REGION Network 1: Green
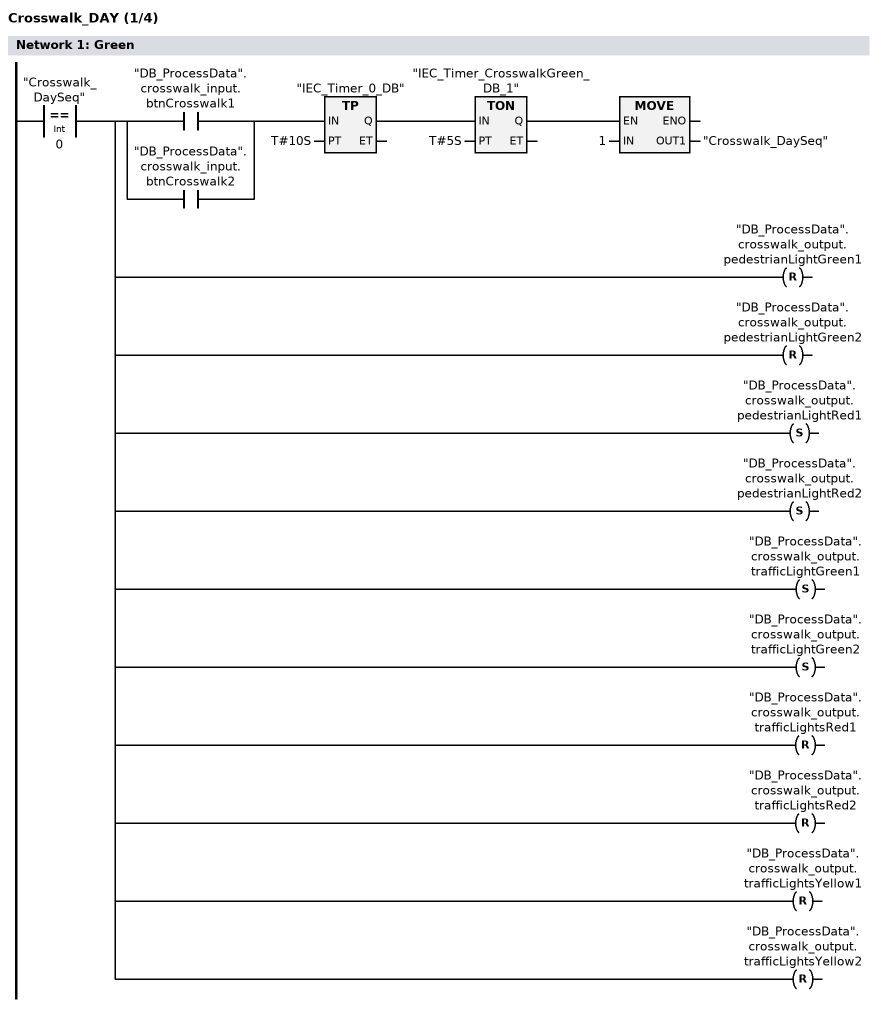
   #_w1 := "Crosswalk_DaySeq" = 0;
   "IEC_Timer_0_DB".TP(IN := #_w1 AND ("DB_ProcessData".crosswalk_input.btnCrosswalk1 OR "DB_ProcessData".crosswalk_input.btnCrosswalk2),
                       PT := T#10S);
   "IEC_Timer_CrosswalkGreen_DB_1".TON(IN := "IEC_Timer_0_DB".Q, PT := T#5S);
   IF "IEC_Timer_CrosswalkGreen_DB_1".Q THEN "Crosswalk_DaySeq" := 1; END_IF;
   IF #_w1 THEN
       "DB_ProcessData".crosswalk_output.pedestrianLightGreen1 := FALSE;
       "DB_ProcessData".crosswalk_output.pedestrianLightGreen2 := FALSE;
       "DB_ProcessData".crosswalk_output.pedestrianLightRed1 := TRUE;
       "DB_ProcessData".crosswalk_output.pedestrianLightRed2 := TRUE;
       "DB_ProcessData".crosswalk_output.trafficLightGreen1 := TRUE;
       "DB_ProcessData".crosswalk_output.trafficLightGreen2 := TRUE;
       "DB_ProcessData".crosswalk_output.trafficLightsRed1 := FALSE;
       "DB_ProcessData".crosswalk_output.trafficLightsRed2 := FALSE;
       "DB_ProcessData".crosswalk_output.trafficLightsYellow1 := FALSE;
       "DB_ProcessData".crosswalk_output.trafficLightsYellow2 := FALSE;
   END_IF;
END_REGION

REGION Network 2: Yellow1
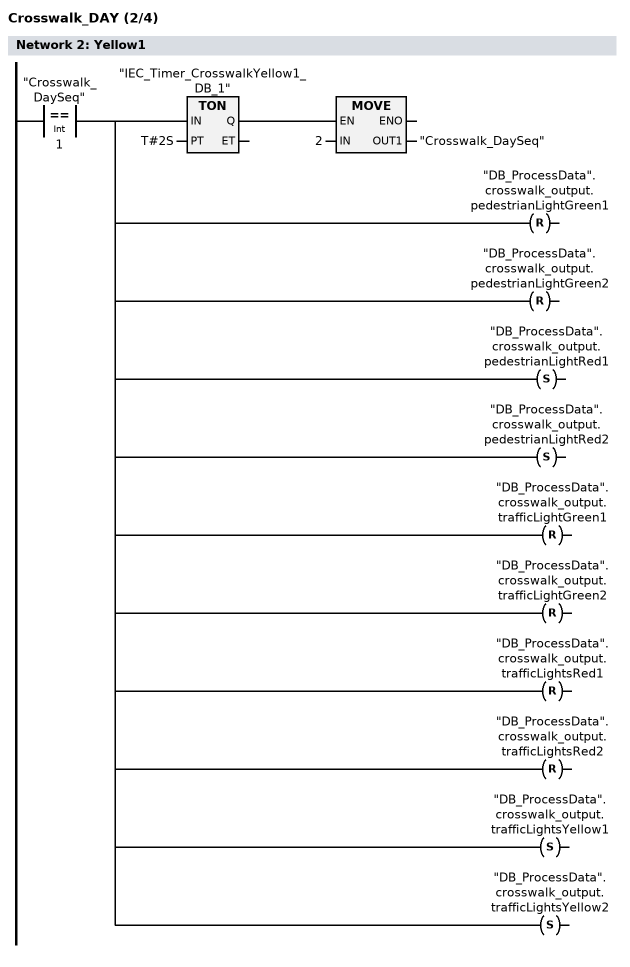
   #_w1 := "Crosswalk_DaySeq" = 1;
   "IEC_Timer_CrosswalkYellow1_DB_1".TON(IN := #_w1, PT := T#2S);
   IF "IEC_Timer_CrosswalkYellow1_DB_1".Q THEN "Crosswalk_DaySeq" := 2; END_IF;
   IF #_w1 THEN
       "DB_ProcessData".crosswalk_output.pedestrianLightGreen1 := FALSE;
       "DB_ProcessData".crosswalk_output.pedestrianLightGreen2 := FALSE;
       "DB_ProcessData".crosswalk_output.pedestrianLightRed1 := TRUE;
       "DB_ProcessData".crosswalk_output.pedestrianLightRed2 := TRUE;
       "DB_ProcessData".crosswalk_output.trafficLightGreen1 := FALSE;
       "DB_ProcessData".crosswalk_output.trafficLightGreen2 := FALSE;
       "DB_ProcessData".crosswalk_output.trafficLightsRed1 := FALSE;
       "DB_ProcessData".crosswalk_output.trafficLightsRed2 := FALSE;
       "DB_ProcessData".crosswalk_output.trafficLightsYellow1 := TRUE;
       "DB_ProcessData".crosswalk_output.trafficLightsYellow2 := TRUE;
   END_IF;
END_REGION

REGION Network 3: Red
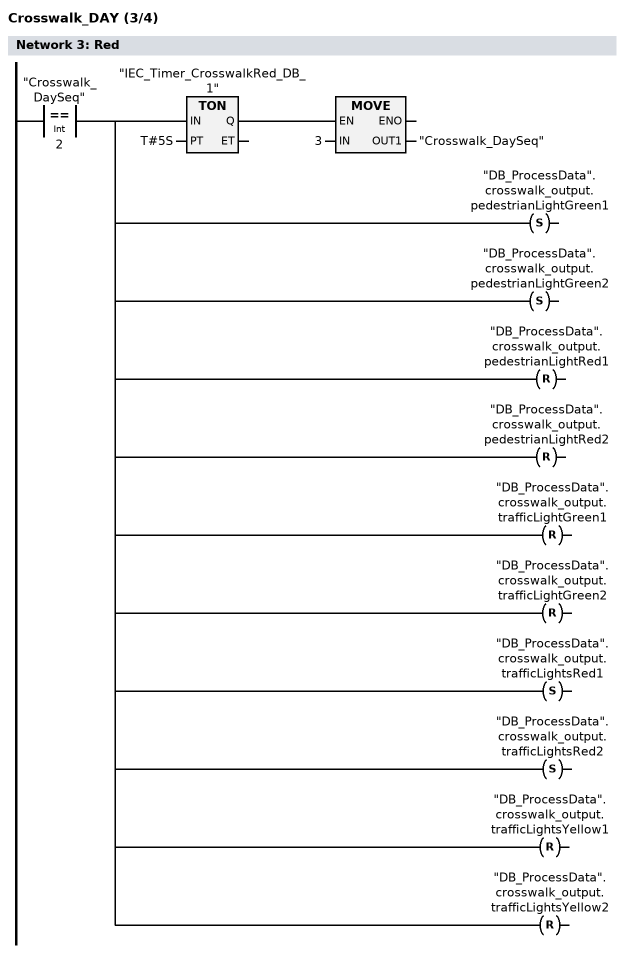
   #_w1 := "Crosswalk_DaySeq" = 2;
   "IEC_Timer_CrosswalkRed_DB_1".TON(IN := #_w1, PT := T#5S);
   IF "IEC_Timer_CrosswalkRed_DB_1".Q THEN "Crosswalk_DaySeq" := 3; END_IF;
   IF #_w1 THEN
       "DB_ProcessData".crosswalk_output.pedestrianLightGreen1 := TRUE;
       "DB_ProcessData".crosswalk_output.pedestrianLightGreen2 := TRUE;
       "DB_ProcessData".crosswalk_output.pedestrianLightRed1 := FALSE;
       "DB_ProcessData".crosswalk_output.pedestrianLightRed2 := FALSE;
       "DB_ProcessData".crosswalk_output.trafficLightGreen1 := FALSE;
       "DB_ProcessData".crosswalk_output.trafficLightGreen2 := FALSE;
       "DB_ProcessData".crosswalk_output.trafficLightsRed1 := TRUE;
       "DB_ProcessData".crosswalk_output.trafficLightsRed2 := TRUE;
       "DB_ProcessData".crosswalk_output.trafficLightsYellow1 := FALSE;
       "DB_ProcessData".crosswalk_output.trafficLightsYellow2 := FALSE;
   END_IF;
END_REGION

REGION Network 4: Yellow2
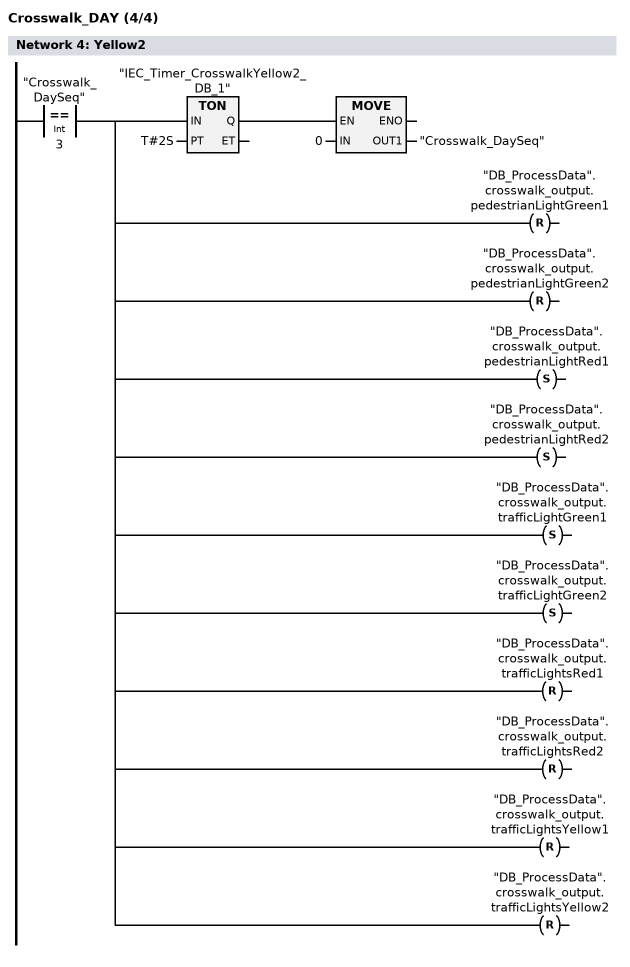
   #_w1 := "Crosswalk_DaySeq" = 3;
   "IEC_Timer_CrosswalkYellow2_DB_1".TON(IN := #_w1, PT := T#2S);
   IF "IEC_Timer_CrosswalkYellow2_DB_1".Q THEN "Crosswalk_DaySeq" := 0; END_IF;
   IF #_w1 THEN
       "DB_ProcessData".crosswalk_output.pedestrianLightGreen1 := FALSE;
       "DB_ProcessData".crosswalk_output.pedestrianLightGreen2 := FALSE;
       "DB_ProcessData".crosswalk_output.pedestrianLightRed1 := TRUE;
       "DB_ProcessData".crosswalk_output.pedestrianLightRed2 := TRUE;
       "DB_ProcessData".crosswalk_output.trafficLightGreen1 := TRUE;
       "DB_ProcessData".crosswalk_output.trafficLightGreen2 := TRUE;
       "DB_ProcessData".crosswalk_output.trafficLightsRed1 := FALSE;
       "DB_ProcessData".crosswalk_output.trafficLightsRed2 := FALSE;
       "DB_ProcessData".crosswalk_output.trafficLightsYellow1 := FALSE;
       "DB_ProcessData".crosswalk_output.trafficLightsYellow2 := FALSE;
   END_IF;
END_REGION
END_FUNCTION

FUNCTION "Crosswalk_NIGHT" : Void   // FC3, LAD
{ S7_Optimized_Access := 'TRUE' }
VERSION : 0.1
   VAR_TEMP   // added for the SCL form of the ladder/FBD networks
      _w1 : Bool;
   END_VAR
BEGIN

REGION Network 1: On
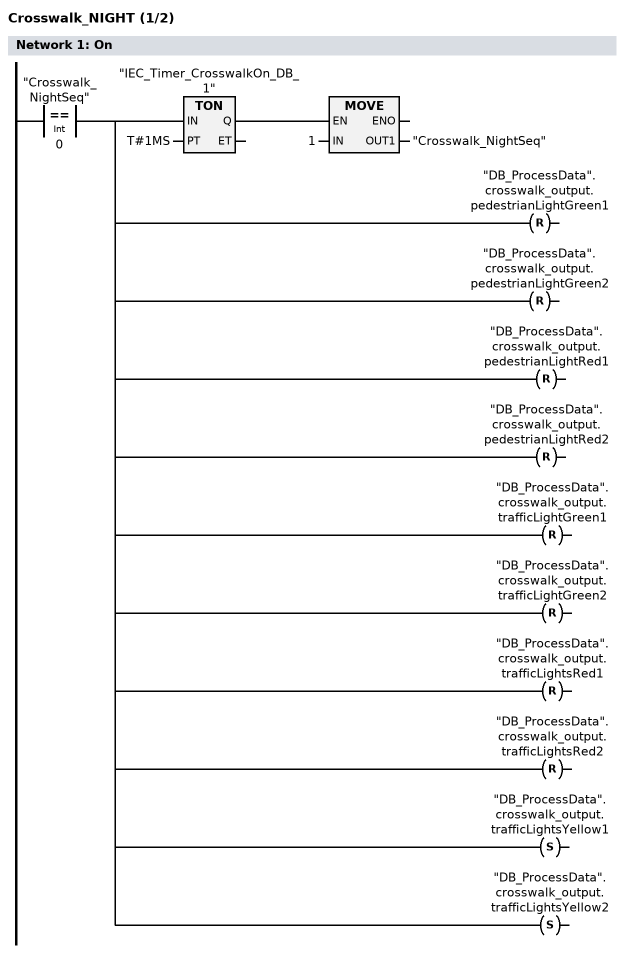
   #_w1 := "Crosswalk_NightSeq" = 0;
   "IEC_Timer_CrosswalkOn_DB_1".TON(IN := #_w1, PT := T#1MS);
   IF "IEC_Timer_CrosswalkOn_DB_1".Q THEN "Crosswalk_NightSeq" := 1; END_IF;
   IF #_w1 THEN
       "DB_ProcessData".crosswalk_output.pedestrianLightGreen1 := FALSE;
       "DB_ProcessData".crosswalk_output.pedestrianLightGreen2 := FALSE;
       "DB_ProcessData".crosswalk_output.pedestrianLightRed1 := FALSE;
       "DB_ProcessData".crosswalk_output.pedestrianLightRed2 := FALSE;
       "DB_ProcessData".crosswalk_output.trafficLightGreen1 := FALSE;
       "DB_ProcessData".crosswalk_output.trafficLightGreen2 := FALSE;
       "DB_ProcessData".crosswalk_output.trafficLightsRed1 := FALSE;
       "DB_ProcessData".crosswalk_output.trafficLightsRed2 := FALSE;
       "DB_ProcessData".crosswalk_output.trafficLightsYellow1 := TRUE;
       "DB_ProcessData".crosswalk_output.trafficLightsYellow2 := TRUE;
   END_IF;
END_REGION

REGION Network 2: Off
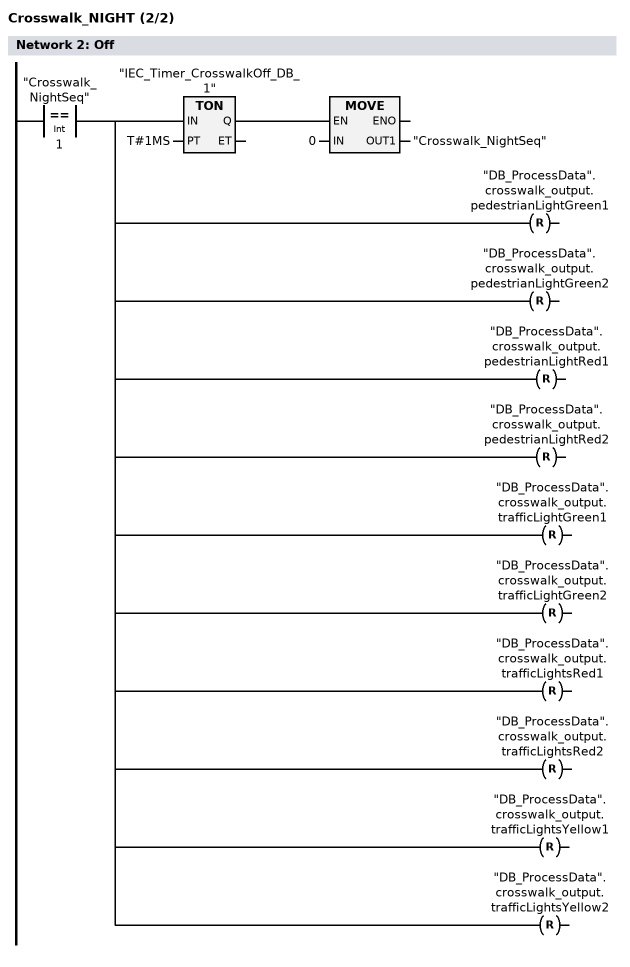
   #_w1 := "Crosswalk_NightSeq" = 1;
   "IEC_Timer_CrosswalkOff_DB_1".TON(IN := #_w1, PT := T#1MS);
   IF "IEC_Timer_CrosswalkOff_DB_1".Q THEN "Crosswalk_NightSeq" := 0; END_IF;
   IF #_w1 THEN
       "DB_ProcessData".crosswalk_output.pedestrianLightGreen1 := FALSE;
       "DB_ProcessData".crosswalk_output.pedestrianLightGreen2 := FALSE;
       "DB_ProcessData".crosswalk_output.pedestrianLightRed1 := FALSE;
       "DB_ProcessData".crosswalk_output.pedestrianLightRed2 := FALSE;
       "DB_ProcessData".crosswalk_output.trafficLightGreen1 := FALSE;
       "DB_ProcessData".crosswalk_output.trafficLightGreen2 := FALSE;
       "DB_ProcessData".crosswalk_output.trafficLightsRed1 := FALSE;
       "DB_ProcessData".crosswalk_output.trafficLightsRed2 := FALSE;
       "DB_ProcessData".crosswalk_output.trafficLightsYellow1 := FALSE;
       "DB_ProcessData".crosswalk_output.trafficLightsYellow2 := FALSE;
   END_IF;
END_REGION
END_FUNCTION

// folder: Regulator

FUNCTION "Regulator_PID" : Void   // FC5, LAD
{ S7_Optimized_Access := 'TRUE' }
VERSION : 0.1
BEGIN

REGION Network 1 (SCL)
   CASE "DB_ProcessData".regulator_input.order OF
       1:
           "Regulator_PV" := "DB_ProcessData".regulator_input.Uc1;
       2:
           "Regulator_PV" := "DB_ProcessData".regulator_input.Uc2;
       ELSE
           "Regulator_PV" := 0;
   END_CASE;

   "Regulator_SetPoint" := 50;
END_REGION

REGION Network 2
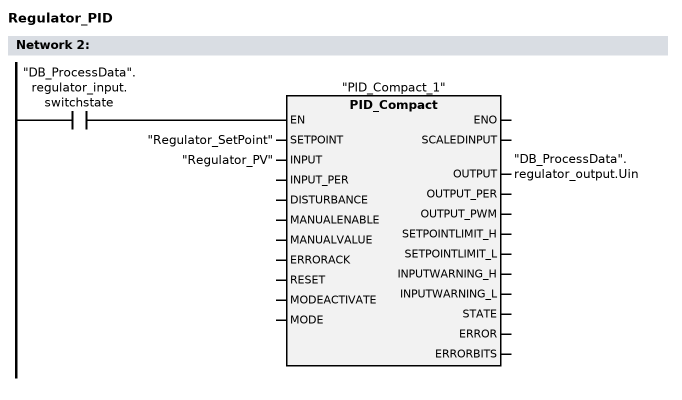
   IF "DB_ProcessData".regulator_input.switchstate THEN
       "PID_Compact_1"(Setpoint := "Regulator_SetPoint",   // PID_Compact
                       Input := "Regulator_PV",
                       Output => "DB_ProcessData".regulator_output.Uin);
   END_IF;
END_REGION
END_FUNCTION

// ===== PLC "R2D2_RESTAPI"  CPU 1212C DC/DC/DC =====

VAR_GLOBAL   // PLC tag table "Default tag table"
   "Clock_Byte" AT %MB0 : Byte;
   "Clock_10Hz" AT %M0.0 : Bool;
   "Clock_5Hz" AT %M0.1 : Bool;
   "Clock_2.5Hz" AT %M0.2 : Bool;
   "Clock_2Hz" AT %M0.3 : Bool;
   "Clock_1.25Hz" AT %M0.4 : Bool;
   "Clock_1Hz" AT %M0.5 : Bool;
   "Clock_0.625Hz" AT %M0.6 : Bool;
   "Clock_0.5Hz" AT %M0.7 : Bool;
   "System_Byte" AT %MB1 : Byte;
   "FirstScan" AT %M1.0 : Bool;
   "DiagStatusUpdate" AT %M1.1 : Bool;
   "AlwaysTRUE" AT %M1.2 : Bool;
   "AlwaysFALSE" AT %M1.3 : Bool;
END_VAR

VAR_GLOBAL   // PLC tag table "Regulator"
   "Regulator_PV" AT %MD100 : Real;
   "Regulator_SetPoint" AT %MD104 : Real;
END_VAR

VAR_GLOBAL   // PLC tag table "CarLight"
   "CarLight_Tag1" AT %I0.0 : Bool;
END_VAR

VAR_GLOBAL   // PLC tag table "Crossroad"
   "Crossroad_Tag_1" AT %M300.0 : Bool;
   "Crossroad_Tag_2" AT %M300.1 : Bool;
   "Crossroad_Tag_3" AT %MW302 : Word;
   "Crossroad_MEM 0" AT %M304.0 : Bool;
   "Crossroad_MEM 1" AT %M304.1 : Bool;
   "Crossroad_MEM 2" AT %M304.2 : Bool;
   "Crossroad_MEM 3" AT %M304.3 : Bool;
   "Crossroad_MEM 5" AT %M304.4 : Bool;
   "Crossroad_MEM 6" AT %M304.5 : Bool;
   "Crossroad_Clock" AT %MW328 : Int;
   "Crossroad_DayModeState" AT %MB305 : USInt;
   "Crossroad_ActualLengthState" AT %MD316 : Time;
   "Crossorad_HoursDayStart" AT %MW320 : Int;
   "Crossroad_HoursDayEnd" AT %MW322 : Int;
   "Crossroad_DayStarts" AT %MW324 : Int;
   "Crossroad_DayEnds" AT %MW326 : Int;
   "Crossroad_S1" AT %MB306 : USInt;
   "Crossroad_S2" AT %MB307 : USInt;
   "Crossroad_S3" AT %MB308 : USInt;
   "Crossroad_S4" AT %MB309 : USInt;
   "Crossroad_S5" AT %MB310 : USInt;
   "Crossroad_S6" AT %MB311 : USInt;
   "Crossroad_S7" AT %MB312 : USInt;
   "Crossroad_S8" AT %MB313 : USInt;
   "Crossroad_S9" AT %MB314 : USInt;
   "Crossroad_Walk_EN" AT %M330.0 : Bool;
END_VAR

VAR_GLOBAL   // PLC tag table "Crosswalk"
   "Crosswalk_CTU_current_value" AT %MW200 : Int;
   "Crosswalk_CTU_reset" AT %M202.0 : Bool;
   "Crosswalk_DayMode" AT %M202.1 : Bool;
   "Crosswalk_NightMode" AT %M202.2 : Bool;
   "Crosswalk_OffMode" AT %M202.3 : Bool;
   "Crosswalk_DaySeq" AT %MW204 : Int;
   "Crosswalk_NightSeq" AT %MW206 : Int;
END_VAR

TYPE "Crossroad_Input"
   STRUCT
      btnStart : Bool := FALSE;
      btnPause : Bool := FALSE;
      btnStop : Bool := FALSE;
      btnWestCrosswalk1 : Bool := FALSE;
      btnWestCrosswalk2 : Bool := FALSE;
      btnSouthCrosswalk1 : Bool := FALSE;
      btnSouthCrosswalk2 : Bool := FALSE;
      spare1 : DWord := 0;
      spare2 : DWord := 0;
      spare3 : DWord := 0;
      spare4 : DWord := 0;
   END_STRUCT;
END_TYPE

TYPE "Crossroad_Output"
   STRUCT
      crossroadType : Bool := FALSE;
      trafficLightNorth_green : Bool := FALSE;
      trafficLightNorth_yellow : Bool := FALSE;
      trafficLightNorth_red : Bool := FALSE;
      trafficLightSouth_green : Bool := FALSE;
      trafficLightSouth_yellow : Bool := FALSE;
      trafficLightSouth_red : Bool := FALSE;
      trafficLightWest_green : Bool := FALSE;
      trafficLightWest_yellow : Bool := FALSE;
      trafficLightWest_red : Bool := FALSE;
      trafficLightEast_green : Bool := FALSE;
      trafficLightEast_yellow : Bool := FALSE;
      trafficLightEast_red : Bool := FALSE;
      pedestrianSouth1_green : Bool := FALSE;
      pedestrianSouth1_red : Bool := FALSE;
      pedestrianSouth2_green : Bool := FALSE;
      pedestrianSouth2_red : Bool := FALSE;
      pedestrianWest1_green : Bool := FALSE;
      pedestrianWest1_red : Bool := FALSE;
      pedestrianWest2_green : Bool := FALSE;
      pedestrianWest2_red : Bool := FALSE;
      spare1 : DWord := 0;
      spare2 : DWord := 0;
      spare3 : DWord := 0;
      spare4 : DWord := 0;
   END_STRUCT;
END_TYPE

TYPE "Crosswalk_Input"
   STRUCT
      btnStart : Bool := FALSE;
      btnPause : Bool := FALSE;
      btnStop : Bool := FALSE;
      btnCrosswalk1 : Bool := FALSE;
      btnCrosswalk2 : Bool := FALSE;
      spare1 : DWord := 0;
      spare2 : DWord := 0;
      spare3 : DWord := 0;
      spare4 : DWord := 0;
   END_STRUCT;
END_TYPE

TYPE "Crosswalk_Output"
   STRUCT
      crosswalkType : Bool := FALSE;
      trafficLightGreen1 : Bool := FALSE;
      trafficLightsYellow1 : Bool := FALSE;
      trafficLightsRed1 : Bool := FALSE;
      trafficLightGreen2 : Bool := FALSE;
      trafficLightsYellow2 : Bool := FALSE;
      trafficLightsRed2 : Bool := FALSE;
      pedestrianLightGreen1 : Bool := FALSE;
      pedestrianLightRed1 : Bool := FALSE;
      pedestrianLightGreen2 : Bool := FALSE;
      pedestrianLightRed2 : Bool := FALSE;
      spare1 : DWord := 0;
      spare2 : DWord := 0;
      spare3 : DWord := 0;
      spare4 : DWord := 0;
   END_STRUCT;
END_TYPE

TYPE "Regulator_Input"
   STRUCT
      btnReset : Bool := FALSE;
      switchstate : Bool := FALSE;
      order : Int := 1;
      R1 : Real := 0.0;
      R2 : Real := 0.0;
      C1 : Real := 0.0;
      C2 : Real := 0.0;
      Uc1 : Real := 0.0;
      Uc2 : Real := 0.0;
      Td : Real := 0.0;
      Ts : Real := 0.0;
      spare1 : DWord := 0;
      spare2 : DWord := 0;
      spare3 : DWord := 0;
      spare4 : DWord := 0;
   END_STRUCT;
END_TYPE

TYPE "Regulator_Output"
   STRUCT
      Uin : Real := 0.0;
      spare1 : DWord := 0;
      spare2 : DWord := 0;
      spare3 : DWord := 0;
      spare4 : DWord := 0;
   END_STRUCT;
END_TYPE

TYPE "CarLight_Input"
   STRUCT
      btnReset : Bool := FALSE;
      error : Bool := FALSE;
      sensorLight : Bool := FALSE;
      sensorConnectorConnected : Bool := FALSE;
      result : Bool := FALSE;
      spare1 : DWord := 0;
      spare2 : DWord := 0;
      spare3 : DWord := 0;
      spare4 : DWord := 0;
   END_STRUCT;
END_TYPE

TYPE "CarLight_Output"
   STRUCT
      lowBeamLight : Bool := FALSE;
      highBeamLight : Bool := FALSE;
      turnLight : Bool := FALSE;
      spare1 : DWord := 0;
      spare2 : DWord := 0;
      spare3 : DWord := 0;
      spare4 : DWord := 0;
   END_STRUCT;
END_TYPE

// folder: Common

TYPE "typeDiagnostics"
TITLE = typeDiagnostics
// Provides a structure for detailed diagnostics
   STRUCT
      status : Word;   // Status of the block or error identification when error occurred
      subfunctionStatus : DWord;   // Status or return value of called FBs, FCs and system blocks
      stateNumber : DInt;   // State in the state machine of the block where the error occurred
   END_STRUCT;
END_TYPE

// folder: LHTTP

TYPE "LHTTP_typeTLS"
   STRUCT
      validateServerIdentity : Bool;   // Validate the subjectAlternateName in the X.509-V3 certificate of the server to check the identity of the server
      serverCert : UDInt;   // ID of the X.509-V3 certificate (usually a CA certificate) that is used by the TLS client to validate the TLS server authentication. If this parameter is 0, the TLS client uses all (CA) certificates currently loaded in the client certificate store to validate the server authentication.
      clientCert : UDInt;   // ID of own X.509 V3 certificate
   END_STRUCT;
END_TYPE

// folder: (top level)

DATA_BLOCK "DB_ProcessData"   // DB1
{ S7_Optimized_Access := 'TRUE' }
VERSION : 0.1
   VAR
      crossroad_input : "Crossroad_Input";
      crossroad_output : "Crossroad_Output";
      crosswalk_input : "Crosswalk_Input";
      crosswalk_output : "Crosswalk_Output";
      regulator_input : "Regulator_Input";
      regulator_output : "Regulator_Output";
      carlight_input : "CarLight_Input";
      carlight_output : "CarLight_Output";
   END_VAR
BEGIN
END_DATA_BLOCK

DATA_BLOCK "REST_API_DATA"   // DB2
{ S7_Optimized_Access := 'TRUE' }
VERSION : 0.1
   VAR
      DATA : Array[0..10000] of Char;
      REST_API_URL : String := 'http://192.168.1.101:5000/api/data';   // 'http://192.168.1.250:5000/api/data' + 'http://10.129.223.194:5000/api/data' + 'http://192.168.1.250:5000/api/data'
   END_VAR
BEGIN
END_DATA_BLOCK

DATA_BLOCK "LHTTP_PostPut_DB"   // DB13
{ S7_Optimized_Access := 'TRUE' }
AUTHOR : Siemens Industry Online Support
FAMILY : LHTTP
VERSION : 2.2
// stored: InstanceOfName LHTTP_PostPut
"LHTTP_PostPut"
BEGIN
END_DATA_BLOCK

DATA_BLOCK "LHTTP_Get_DB"   // DB14
{ S7_Optimized_Access := 'TRUE' }
AUTHOR : Siemens Industry Online Support
FAMILY : LHTTP
VERSION : 2.2
// stored: InstanceOfName LHTTP_Get
"LHTTP_Get"
BEGIN
END_DATA_BLOCK

// folder: CarLight

DATA_BLOCK "CarLight_SCL_DB"   // DB12
{ S7_Optimized_Access := 'TRUE' }
VERSION : 0.1
// stored: InstanceOfName CarLight_SCL
"CarLight_SCL"
BEGIN
END_DATA_BLOCK

// folder: System blocks/Program resources

DATA_BLOCK "IEC_Counter_0_DB"   // DB2
{ S7_Optimized_Access := 'TRUE' }
AUTHOR : Simatic
FAMILY : IEC
NAME : CNTR
VERSION : 1.0
// stored: InstanceOfName IEC_COUNTER
"IEC_COUNTER"
BEGIN
END_DATA_BLOCK

DATA_BLOCK "IEC_Timer_0_DB"   // DB3
{ S7_Optimized_Access := 'TRUE' }
AUTHOR : Simatic
FAMILY : IEC
NAME : IEC_TMR
VERSION : 1.0
// stored: InstanceOfName IEC_TIMER
"IEC_TIMER"
BEGIN
END_DATA_BLOCK

DATA_BLOCK "IEC_Timer_CrosswalkGreen_DB_1"   // DB4
{ S7_Optimized_Access := 'TRUE' }
AUTHOR : Simatic
FAMILY : IEC
NAME : IEC_TMR
VERSION : 1.0
// stored: InstanceOfName IEC_TIMER
"IEC_TIMER"
BEGIN
END_DATA_BLOCK

DATA_BLOCK "IEC_Timer_CrosswalkYellow1_DB_1"   // DB5
{ S7_Optimized_Access := 'TRUE' }
AUTHOR : Simatic
FAMILY : IEC
NAME : IEC_TMR
VERSION : 1.0
// stored: InstanceOfName IEC_TIMER
"IEC_TIMER"
BEGIN
END_DATA_BLOCK

DATA_BLOCK "IEC_Timer_CrosswalkRed_DB_1"   // DB6
{ S7_Optimized_Access := 'TRUE' }
AUTHOR : Simatic
FAMILY : IEC
NAME : IEC_TMR
VERSION : 1.0
// stored: InstanceOfName IEC_TIMER
"IEC_TIMER"
BEGIN
END_DATA_BLOCK

DATA_BLOCK "IEC_Timer_CrosswalkYellow2_DB_1"   // DB7
{ S7_Optimized_Access := 'TRUE' }
AUTHOR : Simatic
FAMILY : IEC
NAME : IEC_TMR
VERSION : 1.0
// stored: InstanceOfName IEC_TIMER
"IEC_TIMER"
BEGIN
END_DATA_BLOCK

DATA_BLOCK "IEC_Timer_CrosswalkOn_DB_1"   // DB8
{ S7_Optimized_Access := 'TRUE' }
AUTHOR : Simatic
FAMILY : IEC
NAME : IEC_TMR
VERSION : 1.0
// stored: InstanceOfName IEC_TIMER
"IEC_TIMER"
BEGIN
END_DATA_BLOCK

DATA_BLOCK "IEC_Timer_CrosswalkOff_DB_1"   // DB9
{ S7_Optimized_Access := 'TRUE' }
AUTHOR : Simatic
FAMILY : IEC
NAME : IEC_TMR
VERSION : 1.0
// stored: InstanceOfName IEC_TIMER
"IEC_TIMER"
BEGIN
END_DATA_BLOCK

DATA_BLOCK "IEC_Timer_CrossroadCycle_DB_1"   // DB10
{ S7_Optimized_Access := 'TRUE' }
AUTHOR : Simatic
FAMILY : IEC
NAME : IEC_TMR
VERSION : 1.0
// stored: InstanceOfName IEC_TIMER
"IEC_TIMER"
BEGIN
END_DATA_BLOCK

// folder: (top level)

ORGANIZATION_BLOCK "Main"   // OB1, LAD, ProgramCycle
TITLE = "Main Program Sweep (Cycle)"
{ S7_Optimized_Access := 'TRUE' }
VERSION : 0.1
   VAR_INPUT
      Initial_Call : Bool;   // Initial call of this OB
      Remanence : Bool;   // =True, if remanent data are available
   END_VAR
BEGIN

REGION Network 1: REST API - POST & GET
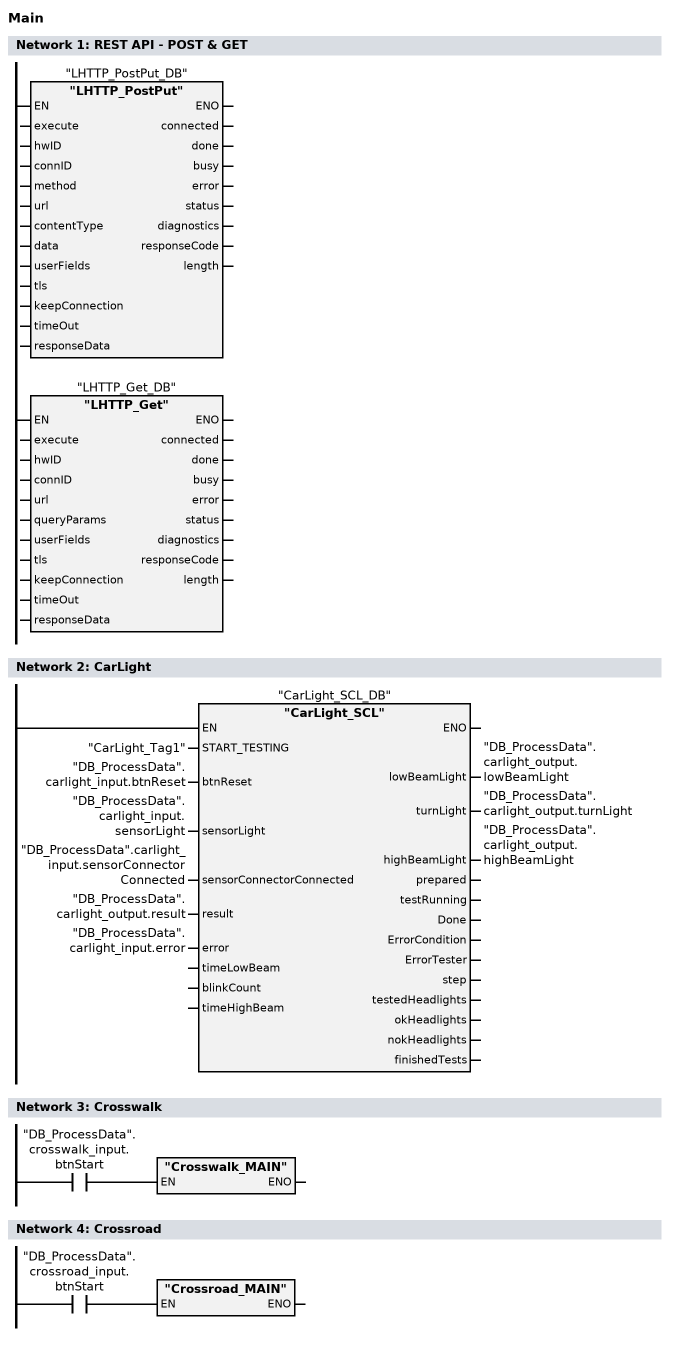
   RUNG wire#powerrail
      "LHTTP_PostPut_DB"(execute :=, hwID :=, connID :=, method :=, url :=, contentType :=, data :=, userFields :=, tls :=, keepConnection :=, timeOut :=, responseData :=, connected =>, done =>, busy =>, error =>, status =>, diagnostics =>, responseCode =>, length =>)
   END_RUNG
   RUNG wire#powerrail
      "LHTTP_Get_DB"(execute :=, hwID :=, connID :=, url :=, queryParams :=, userFields :=, tls :=, keepConnection :=, timeOut :=, responseData :=, connected =>, done =>, busy =>, error =>, status =>, diagnostics =>, responseCode =>, length =>)
   END_RUNG
   // the same network as SCL:
   "LHTTP_PostPut_DB"();   // "LHTTP_PostPut"
   "LHTTP_Get_DB"();   // "LHTTP_Get"
END_REGION

REGION Network 2: CarLight
   RUNG wire#powerrail
      "CarLight_SCL_DB"(START_TESTING := "CarLight_Tag1", btnReset := "DB_ProcessData".carlight_input.btnReset, sensorLight := "DB_ProcessData".carlight_input.sensorLight, sensorConnectorConnected := "DB_ProcessData".carlight_input.sensorConnectorConnected, result := "DB_ProcessData".carlight_output.result, error := "DB_ProcessData".carlight_input.error, timeLowBeam :=, blinkCount :=, timeHighBeam :=, lowBeamLight => "DB_ProcessData".carlight_output.lowBeamLight, turnLight => "DB_ProcessData".carlight_output.turnLight, highBeamLight => "DB_ProcessData".carlight_output.highBeamLight, prepared =>, testRunning =>, Done =>, ErrorCondition =>, ErrorTester =>, "step" =>, testedHeadlights =>, okHeadlights =>, nokHeadlights =>, finishedTests =>)
   END_RUNG
   // the same network as SCL:
   "CarLight_SCL_DB"(START_TESTING := "CarLight_Tag1",   // "CarLight_SCL"
                     btnReset := "DB_ProcessData".carlight_input.btnReset,
                     sensorLight := "DB_ProcessData".carlight_input.sensorLight,
                     sensorConnectorConnected := "DB_ProcessData".carlight_input.sensorConnectorConnected,
                     result := "DB_ProcessData".carlight_output.result,
                     error := "DB_ProcessData".carlight_input.error,
                     lowBeamLight => "DB_ProcessData".carlight_output.lowBeamLight,
                     turnLight => "DB_ProcessData".carlight_output.turnLight,
                     highBeamLight => "DB_ProcessData".carlight_output.highBeamLight);
END_REGION

REGION Network 3: Crosswalk
   RUNG wire#powerrail
      Contact( "DB_ProcessData".crosswalk_input.btnStart )
      "Crosswalk_MAIN"()
   END_RUNG
   // the same network as SCL:
   IF "DB_ProcessData".crosswalk_input.btnStart THEN "Crosswalk_MAIN"(); END_IF;
END_REGION

REGION Network 4: Crossroad
   RUNG wire#powerrail
      Contact( "DB_ProcessData".crossroad_input.btnStart )
      "Crossroad_MAIN"()
   END_RUNG
   // the same network as SCL:
   IF "DB_ProcessData".crossroad_input.btnStart THEN "Crossroad_MAIN"(); END_IF;
END_REGION
END_ORGANIZATION_BLOCK

ORGANIZATION_BLOCK "CyclicInterrupt"   // OB30, LAD, CyclicInterrupt
{ S7_Optimized_Access := 'TRUE' }
VERSION : 0.1
   VAR_INPUT
      Initial_Call : Bool;   // Initial call of this OB
      Event_Count : Int;   // Events discarded
   END_VAR
BEGIN

REGION Network 1: Regulator
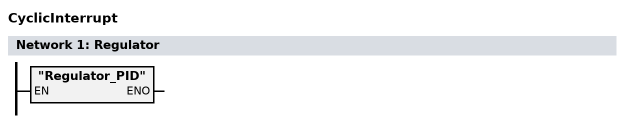
   RUNG wire#powerrail
      "Regulator_PID"()
   END_RUNG
   // the same network as SCL:
   "Regulator_PID"();
END_REGION
END_ORGANIZATION_BLOCK

ORGANIZATION_BLOCK "Startup"   // OB100, LAD, Startup
TITLE = "Complete Restart"
{ S7_Optimized_Access := 'TRUE' }
VERSION : 0.1
   VAR_INPUT
      LostRetentive : Bool;   // True if retentive data are lost
      LostRTC : Bool;   // True if date and time are lost
   END_VAR
BEGIN

REGION Network 1 (SCL)
   // Communication 


   // Crossroad
   "Crossorad_HoursDayStart" := 0;
   "Crossroad_HoursDayEnd" := 2400;
   "Crossroad_DayStarts" := 500;
   "Crossroad_DayEnds" := 2200;
   "Crossroad_S1" := 1;
   "Crossroad_S2" := 2;
   "Crossroad_S3" := 3;
   "Crossroad_S4" := 4;
   "Crossroad_S5" := 5;
   "Crossroad_S6" := 6;
   "Crossroad_S7" := 7;
   "Crossroad_S8" := 8;
   "Crossroad_S9" := 9;


   // Crosswalk


   // Regulaotr


   // CarLight
END_REGION
END_ORGANIZATION_BLOCK

// folder: CarLight

FUNCTION_BLOCK "CarLight_SCL"   // FB1, SCL
{ S7_Optimized_Access := 'TRUE' }
VERSION : 0.1
   VAR_INPUT
      START_TESTING : Bool;
      btnReset : Bool;
      sensorLight : Bool;
      sensorConnectorConnected : Bool;
      result : Bool;
      error : Bool;
      timeLowBeam : Time;
      blinkCount : Int;
      timeHighBeam : Time;
   END_VAR
   VAR_OUTPUT
      lowBeamLight : Bool;
      turnLight : Bool;
      highBeamLight : Bool;
      prepared : Bool;
      testRunning : Bool;
      Done : Bool;
      ErrorCondition : Bool;
      ErrorTester : Bool;
      "step" : Int;
      testedHeadlights : DInt;
      okHeadlights : DInt;
      nokHeadlights : DInt;
      finishedTests : DInt;
   END_VAR
   VAR
      state : Int;
      ready : Bool;
      start_old : Bool;
      start_rise : Bool;
      conditionsErrorLatched : Bool;
      testerErrorLatched : Bool;
      blinkTarget : Int;
      blinkIndex : Int;
      resultStored : Bool;
      testerResponseSeenTrue : Bool;
      tonLowBeam : TON_TIME;
      tonBlinkOn : TON_TIME;
      tonBlinkOff : TON_TIME;
      tonHighBeam : TON_TIME;
      tonAll : TON_TIME;
      tonTesterResponse : TON_TIME;
   END_VAR
BEGIN
   // ---------------------------------------------------------------------
   // Helper signals
   // ---------------------------------------------------------------------
   #ready := #sensorLight AND #sensorConnectorConnected;

   IF #blinkCount < 1 THEN
       #blinkTarget := 1;
   ELSE
       #blinkTarget := #blinkCount;
   END_IF;

   #start_rise := #START_TESTING AND NOT #start_old;
   #start_old := #START_TESTING;


   // ---------------------------------------------------------------------
   // RESET process (counters are NOT cleared)
   // ---------------------------------------------------------------------
   IF #btnReset THEN
       #state := 0;
       #conditionsErrorLatched := FALSE;
       #testerErrorLatched := FALSE;
       #blinkIndex := 0;
       #resultStored := FALSE;
       #testerResponseSeenTrue := FALSE;
   END_IF;


   // ---------------------------------------------------------------------
   // Loss of required conditions during test
   // ---------------------------------------------------------------------
   IF ((#state >= 20) AND (#state <= 55)) AND (NOT #ready) THEN
       #state := 0;
       #conditionsErrorLatched := TRUE;
       #blinkIndex := 0;
       #resultStored := FALSE;
       #testerResponseSeenTrue := FALSE;
   END_IF;


   // ---------------------------------------------------------------------
   // Tester error – immediate NOK termination
   // ---------------------------------------------------------------------
   IF ((#state >= 20) AND (#state <= 55)) AND #error THEN

       #testerErrorLatched := TRUE;

       IF NOT #resultStored THEN
           #testedHeadlights := #testedHeadlights + 1;
           #nokHeadlights := #nokHeadlights + 1;
           #resultStored := TRUE;
       END_IF;

       #blinkIndex := 0;
       #testerResponseSeenTrue := FALSE;

       #state := 70;

   END_IF;


   // ---------------------------------------------------------------------
   // State machine
   // ---------------------------------------------------------------------
   CASE #state OF


           // ==============================================================
           // 0 - IDLE
           // ==============================================================
       0:

           #lowBeamLight := FALSE;
           #turnLight := FALSE;
           #highBeamLight := FALSE;

           #tonLowBeam(IN := FALSE,
                     PT := #timeLowBeam);
           #tonBlinkOn(IN := FALSE,
                       PT := T#1s);
           #tonBlinkOff(IN := FALSE,
                        PT := T#1s);
           #tonHighBeam(IN := FALSE,
                     PT := #timeHighBeam);
           #tonAll(IN := FALSE,
                   PT := T#5s);
           #tonTesterResponse(IN := FALSE,
                              PT := T#1s);

           IF #start_rise THEN

               IF #ready AND (NOT #error) THEN

                   #conditionsErrorLatched := FALSE;
                   #testerErrorLatched := FALSE;
                   #blinkIndex := 0;
                   #resultStored := FALSE;
                   #testerResponseSeenTrue := FALSE;

                   #state := 20;

               ELSE

                   IF NOT #ready THEN
                       #conditionsErrorLatched := TRUE;
                   END_IF;

                   IF #error THEN
                       #testerErrorLatched := TRUE;
                   END_IF;

               END_IF;

           END_IF;


           // ==============================================================
           // 20 - LOW BEAM
           // ==============================================================
       20:

           #lowBeamLight := TRUE;
           #turnLight := FALSE;
           #highBeamLight := FALSE;

           #tonLowBeam(IN := TRUE,
                     PT := #timeLowBeam);
           #tonBlinkOn(IN := FALSE,
                       PT := T#1s);
           #tonBlinkOff(IN := FALSE,
                        PT := T#1s);
           #tonHighBeam(IN := FALSE,
                     PT := #timeHighBeam);
           #tonAll(IN := FALSE,
                   PT := T#5s);
           #tonTesterResponse(IN := FALSE,
                              PT := T#1s);

           IF #tonLowBeam.Q THEN
               #blinkIndex := 0;
               #state := 30;
           END_IF;


           // ==============================================================
           // 30 - TURN SIGNAL ON
           // ==============================================================
       30:

           #lowBeamLight := FALSE;
           #turnLight := TRUE;
           #highBeamLight := FALSE;

           #tonLowBeam(IN := FALSE,
                     PT := #timeLowBeam);
           #tonBlinkOn(IN := TRUE,
                       PT := T#1s);
           #tonBlinkOff(IN := FALSE,
                        PT := T#1s);
           #tonHighBeam(IN := FALSE,
                     PT := #timeHighBeam);
           #tonAll(IN := FALSE,
                   PT := T#5s);
           #tonTesterResponse(IN := FALSE,
                              PT := T#1s);

           IF #tonBlinkOn.Q THEN
               #state := 31;
           END_IF;


           // ==============================================================
           // 31 - TURN SIGNAL OFF
           // ==============================================================
       31:

           #lowBeamLight := FALSE;
           #turnLight := FALSE;
           #highBeamLight := FALSE;

           #tonLowBeam(IN := FALSE,
                     PT := #timeLowBeam);
           #tonBlinkOn(IN := FALSE,
                       PT := T#1s);
           #tonBlinkOff(IN := TRUE,
                        PT := T#1s);
           #tonHighBeam(IN := FALSE,
                     PT := #timeHighBeam);
           #tonAll(IN := FALSE,
                   PT := T#5s);
           #tonTesterResponse(IN := FALSE,
                              PT := T#1s);

           IF #tonBlinkOff.Q THEN

               #blinkIndex := #blinkIndex + 1;

               IF #blinkIndex < #blinkTarget THEN
                   #state := 30;
               ELSE
                   #state := 40;
               END_IF;

           END_IF;


           // ==============================================================
           // 40 - HIGH BEAM
           // ==============================================================
       40:

           #lowBeamLight := FALSE;
           #turnLight := FALSE;
           #highBeamLight := TRUE;

           #tonLowBeam(IN := FALSE,
                     PT := #timeLowBeam);
           #tonBlinkOn(IN := FALSE,
                       PT := T#1s);
           #tonBlinkOff(IN := FALSE,
                        PT := T#1s);
           #tonHighBeam(IN := TRUE,
                     PT := #timeHighBeam);
           #tonAll(IN := FALSE,
                   PT := T#5s);
           #tonTesterResponse(IN := FALSE,
                              PT := T#1s);

           IF #tonHighBeam.Q THEN
               #state := 50;
           END_IF;


           // ==============================================================
           // 50 - ALL LIGHTS (5 seconds)
           // ==============================================================
       50:

           #lowBeamLight := TRUE;
           #turnLight := TRUE;
           #highBeamLight := TRUE;

           #tonLowBeam(IN := FALSE,
                     PT := #timeLowBeam);
           #tonBlinkOn(IN := FALSE,
                       PT := T#1s);
           #tonBlinkOff(IN := FALSE,
                        PT := T#1s);
           #tonHighBeam(IN := FALSE,
                     PT := #timeHighBeam);
           #tonAll(IN := TRUE,
                   PT := T#5s);
           #tonTesterResponse(IN := FALSE,
                              PT := T#1s);

           IF #tonAll.Q THEN
               #testerResponseSeenTrue := FALSE;
               #state := 55;
           END_IF;


           // ==============================================================
           // 55 - WAIT 1 s FOR RESULT
           // ==============================================================
       55:

           #lowBeamLight := FALSE;
           #turnLight := FALSE;
           #highBeamLight := FALSE;

           #tonLowBeam(IN := FALSE,
                     PT := #timeLowBeam);
           #tonBlinkOn(IN := FALSE,
                       PT := T#1s);
           #tonBlinkOff(IN := FALSE,
                        PT := T#1s);
           #tonHighBeam(IN := FALSE,
                     PT := #timeHighBeam);
           #tonAll(IN := FALSE,
                   PT := T#5s);
           #tonTesterResponse(IN := TRUE,
                              PT := T#1s);

           IF #result THEN
               #testerResponseSeenTrue := TRUE;
           END_IF;

           IF #tonTesterResponse.Q THEN

               IF NOT #resultStored THEN

                   #testedHeadlights := #testedHeadlights + 1;

                   IF #testerResponseSeenTrue THEN
                       #okHeadlights := #okHeadlights + 1;
                   ELSE
                       #nokHeadlights := #nokHeadlights + 1;
                   END_IF;

                   #resultStored := TRUE;

               END_IF;

               #finishedTests := #finishedTests + 1;

               #state := 60;

           END_IF;


           // ==============================================================
           // 60 - FINISHED
           // ==============================================================
       60:

           #lowBeamLight := FALSE;
           #turnLight := FALSE;
           #highBeamLight := FALSE;

           IF #start_rise THEN

               IF #ready AND (NOT #error) THEN

                   #conditionsErrorLatched := FALSE;
                   #testerErrorLatched := FALSE;
                   #blinkIndex := 0;
                   #resultStored := FALSE;
                   #testerResponseSeenTrue := FALSE;

                   #state := 20;

               END_IF;

           END_IF;


           // ==============================================================
           // 70 - TESTER ERROR
           // ==============================================================
       70:

           #lowBeamLight := FALSE;
           #turnLight := FALSE;
           #highBeamLight := FALSE;

           IF #start_rise THEN

               IF #ready AND (NOT #error) THEN

                   #conditionsErrorLatched := FALSE;
                   #testerErrorLatched := FALSE;
                   #blinkIndex := 0;
                   #resultStored := FALSE;
                   #testerResponseSeenTrue := FALSE;

                   #state := 20;

               END_IF;

           END_IF;

       ELSE

           #state := 0;

   END_CASE;


   // ---------------------------------------------------------------------
   // State outputs
   // ---------------------------------------------------------------------
   #testRunning := (#state >= 20) AND (#state <= 55);

   #prepared := #ready AND (NOT #error) AND
   ((#state = 0) OR (#state = 60) OR (#state = 70));

   #Done := (#state = 60);

   #ErrorCondition := #conditionsErrorLatched;
   #ErrorTester := #testerErrorLatched;

   #step := #state;
END_FUNCTION_BLOCK

// folder: Common

FUNCTION "IsIPAddress" : Bool   // FC1, SCL
TITLE = IsIPAddress
{ S7_Optimized_Access := 'TRUE' }
VERSION : 0.1
// Evaluates whether a given String contains a valid IP address
   VAR_INPUT
      address : String;   // Address to be evaluated
   END_VAR
   VAR_OUTPUT
      ipAddress : IP_V4;   // Parsed IP address if passed address is IP address
   END_VAR
   VAR_TEMP
      tempAddress : String;   // Passed address
      tempOctet : String;   // Current octet
      tempIndex : DInt;   // Index for loop
      tempPos : Int;   // Position of found separator
      tempNum : Int;   // Converted octet
      tempIp : IP_V4;   // Parsed IP address
   END_VAR
   // Ret_Val : Return value
   VAR CONSTANT
      MAX_VALUE : USInt := 255;   // Max. valid value of octet
      NUM_OCTETS : DInt := 4;   // Number of octets
      CHAR_ZERO : Char := '0';   // ASCII character '0'
   END_VAR
BEGIN
   REGION BLOCK INFO HEADER
     //===============================================================================
     // SIEMENS / (c)Copyright 2024
     //-------------------------------------------------------------------------------
     // Title:        IsIPAddress
     // Function:     Evaluates whether a given String contains a valid IP address
     // Library:      --
     // Author:       Siemens Industry Online Support
     // Tested with:  CPU 1515-2 PN V3.1
     // Engineering:  TIA Portal V17
     // Restrictions: --
     // Requirements: S7-1200 with firmware V4.4 or higher
     //               S7-1500 with firmware V2.0 or higher
     //-------------------------------------------------------------------------------
     // Change log table:
     // Version  | Date       | Expert in charge       | Changes applied
     //-------------------------------------------------------------------------------
     // 01.00.00 | 2024-02-12 | Online Support         | First released version
     //===============================================================================
   END_REGION

   #tempAddress := #address;
   #IsIPAddress := FALSE; // Will be overwritten if IP address is detected
   #ipAddress := #tempIp; // Zero output parameter

   FOR #tempIndex := 1 TO #NUM_OCTETS DO
     #tempPos := FIND(IN1 := #tempAddress, IN2 := '.'); // Find separator

     IF (#tempPos > 0 OR #tempIndex = #NUM_OCTETS) // Separator found with exception of last octet
       AND NOT (#tempPos > 0 AND #tempIndex = #NUM_OCTETS) // No separator found in last octet
       AND #tempPos <= 4 // 3  characters or less
     THEN
       IF #tempIndex < #NUM_OCTETS THEN // First three octets
         #tempOctet := LEFT(IN := #tempAddress, L := #tempPos - 1);
       ELSE// Last octet
         #tempOctet := #tempAddress;
       END_IF;

       STRG_VAL(IN := #tempOctet,
                FORMAT := 0,
                P := 1,
                OUT => #tempNum);

       IF #tempNum >= 0 AND #tempNum <= #MAX_VALUE // Within 0 and 255
         AND NOT (#tempNum = 0 AND #tempIndex = 1) // Not 0 in first octet
         AND NOT (#tempNum = 0 AND #tempOctet[1] <> #CHAR_ZERO) // Not 0 because of invalid character
       THEN
         #tempIp.ADDR[#tempIndex] := INT_TO_BYTE(#tempNum);
         #tempAddress := RIGHT(IN := #tempAddress, L := LEN(#tempAddress) - #tempPos); // Remove evaluated octet
       ELSE // Address is not IP address
         EXIT;
       END_IF;
     ELSE // Address is not IP address
       EXIT;
     END_IF;

     IF #tempIndex = #NUM_OCTETS THEN // End of loop reached, address is IP address
       #ipAddress := #tempIp;
       #IsIPAddress := true;
     END_IF;
   END_FOR;
END_FUNCTION

// folder: Crossroad

FUNCTION "Crossroad_MAIN" : Void   // FC4, LAD
{ S7_Optimized_Access := 'TRUE' }
VERSION : 0.1
   VAR_TEMP   // added for the SCL form of the ladder/FBD networks
      _w1 : Bool;
      _w2 : Bool;
      _w3 : Bool;
      _w4 : Bool;
   END_VAR
BEGIN

REGION Network 1: Time based decision process
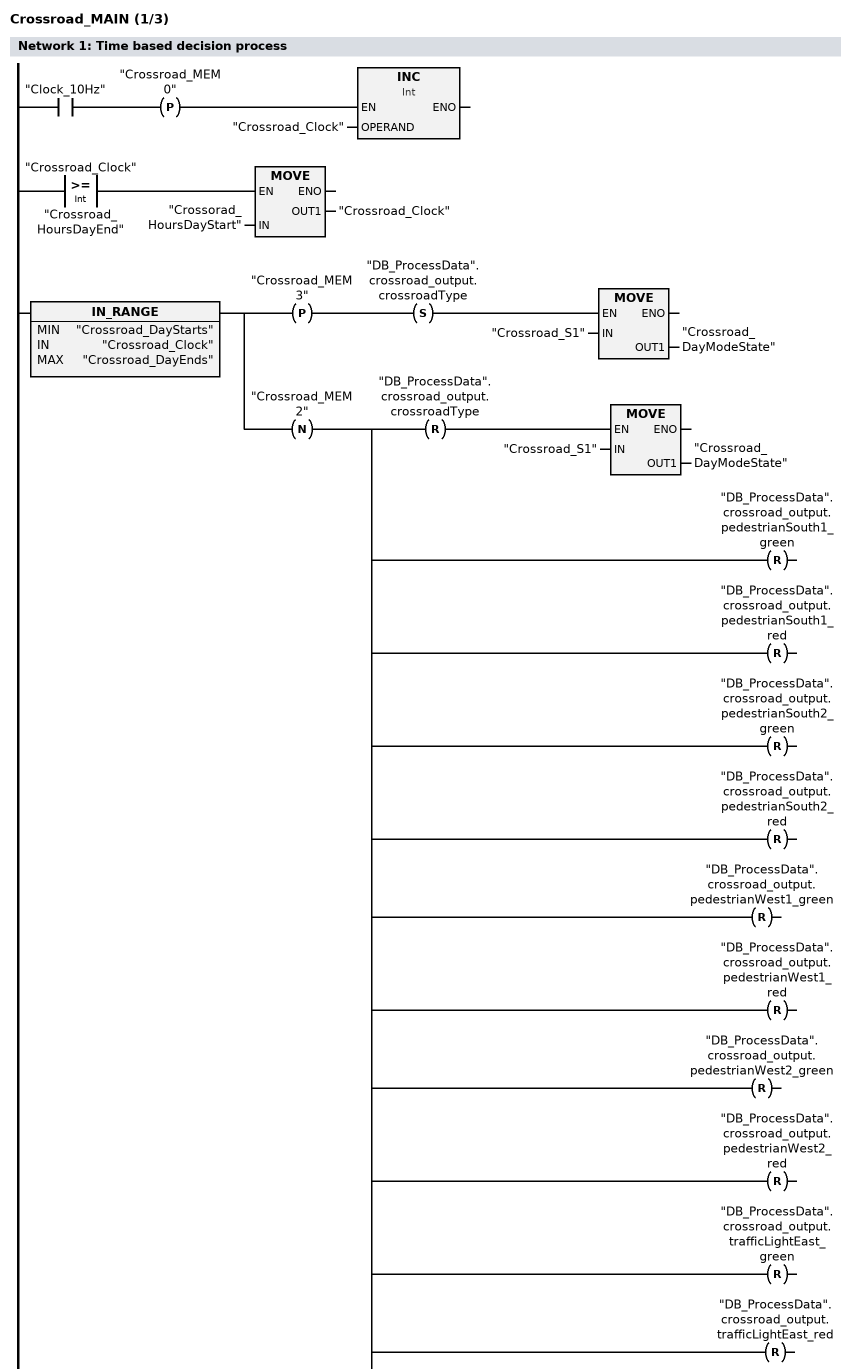
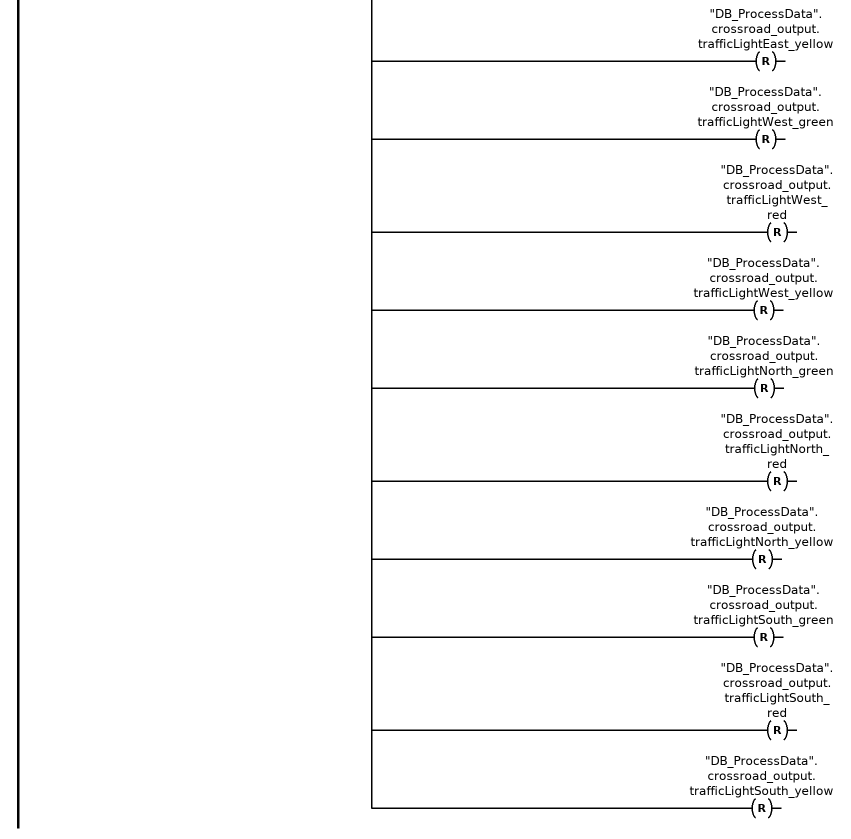
   RUNG wire#powerrail
      Contact( "Clock_10Hz" )
      P_Trig( "Crossroad_MEM 0" )
      { S7_Templates := "DestType := Int" } Inc( "Crossroad_Clock" )
   END_RUNG
   RUNG wire#powerrail
      { S7_Templates := "SrcType := Int" } GE_Contact(in1 := "Crossroad_Clock", in2 := "Crossroad_HoursDayEnd")
      Move(in := "Crossorad_HoursDayStart", out1 => "Crossroad_Clock")
   END_RUNG
   RUNG wire#powerrail
      { S7_Templates := "SrcType := Int" } InRange(min := "Crossroad_DayStarts", in := "Crossroad_Clock", max := "Crossroad_DayEnds")
      wire#w1
      P_Trig( "Crossroad_MEM 3" )
      S_Coil( "DB_ProcessData".crossroad_output.crossroadType )
      Move(in := "Crossroad_S1", out1 => "Crossroad_DayModeState")
   END_RUNG
   RUNG wire#w1
      N_Trig( "Crossroad_MEM 2" )
      wire#w2
      R_Coil( "DB_ProcessData".crossroad_output.crossroadType )
      Move(in := "Crossroad_S1", out1 => "Crossroad_DayModeState")
   END_RUNG
   RUNG wire#w2
      R_Coil( "DB_ProcessData".crossroad_output.pedestrianSouth1_green )
   END_RUNG
   RUNG wire#w2
      R_Coil( "DB_ProcessData".crossroad_output.pedestrianSouth1_red )
   END_RUNG
   RUNG wire#w2
      R_Coil( "DB_ProcessData".crossroad_output.pedestrianSouth2_green )
   END_RUNG
   RUNG wire#w2
      R_Coil( "DB_ProcessData".crossroad_output.pedestrianSouth2_red )
   END_RUNG
   RUNG wire#w2
      R_Coil( "DB_ProcessData".crossroad_output.pedestrianWest1_green )
   END_RUNG
   RUNG wire#w2
      R_Coil( "DB_ProcessData".crossroad_output.pedestrianWest1_red )
   END_RUNG
   RUNG wire#w2
      R_Coil( "DB_ProcessData".crossroad_output.pedestrianWest2_green )
   END_RUNG
   RUNG wire#w2
      R_Coil( "DB_ProcessData".crossroad_output.pedestrianWest2_red )
   END_RUNG
   RUNG wire#w2
      R_Coil( "DB_ProcessData".crossroad_output.trafficLightEast_green )
   END_RUNG
   RUNG wire#w2
      R_Coil( "DB_ProcessData".crossroad_output.trafficLightEast_red )
   END_RUNG
   RUNG wire#w2
      R_Coil( "DB_ProcessData".crossroad_output.trafficLightEast_yellow )
   END_RUNG
   RUNG wire#w2
      R_Coil( "DB_ProcessData".crossroad_output.trafficLightWest_green )
   END_RUNG
   RUNG wire#w2
      R_Coil( "DB_ProcessData".crossroad_output.trafficLightWest_red )
   END_RUNG
   RUNG wire#w2
      R_Coil( "DB_ProcessData".crossroad_output.trafficLightWest_yellow )
   END_RUNG
   RUNG wire#w2
      R_Coil( "DB_ProcessData".crossroad_output.trafficLightNorth_green )
   END_RUNG
   RUNG wire#w2
      R_Coil( "DB_ProcessData".crossroad_output.trafficLightNorth_red )
   END_RUNG
   RUNG wire#w2
      R_Coil( "DB_ProcessData".crossroad_output.trafficLightNorth_yellow )
   END_RUNG
   RUNG wire#w2
      R_Coil( "DB_ProcessData".crossroad_output.trafficLightSouth_green )
   END_RUNG
   RUNG wire#w2
      R_Coil( "DB_ProcessData".crossroad_output.trafficLightSouth_red )
   END_RUNG
   RUNG wire#w2
      R_Coil( "DB_ProcessData".crossroad_output.trafficLightSouth_yellow )
   END_RUNG
   // the same network as SCL:
   #_w1 := "Clock_10Hz" AND NOT "Crossroad_MEM 0";   // rising edge
   "Crossroad_MEM 0" := "Clock_10Hz";
   IF #_w1 THEN "Crossroad_Clock" := "Crossroad_Clock" + 1; END_IF;
   IF "Crossroad_Clock" >= "Crossroad_HoursDayEnd" THEN
       "Crossroad_Clock" := "Crossorad_HoursDayStart";
   END_IF;
   #_w2 := ("Crossroad_DayStarts" <= "Crossroad_Clock") AND ("Crossroad_Clock" <= "Crossroad_DayEnds");
   #_w3 := #_w2 AND NOT "Crossroad_MEM 3";   // rising edge
   "Crossroad_MEM 3" := #_w2;
   IF #_w3 THEN
       "DB_ProcessData".crossroad_output.crossroadType := TRUE;
       "Crossroad_DayModeState" := "Crossroad_S1";
   END_IF;
   #_w4 := NOT #_w2 AND "Crossroad_MEM 2";   // falling edge
   "Crossroad_MEM 2" := #_w2;
   IF #_w4 THEN
       "DB_ProcessData".crossroad_output.crossroadType := FALSE;
       "Crossroad_DayModeState" := "Crossroad_S1";
       "DB_ProcessData".crossroad_output.pedestrianSouth1_green := FALSE;
       "DB_ProcessData".crossroad_output.pedestrianSouth1_red := FALSE;
       "DB_ProcessData".crossroad_output.pedestrianSouth2_green := FALSE;
       "DB_ProcessData".crossroad_output.pedestrianSouth2_red := FALSE;
       "DB_ProcessData".crossroad_output.pedestrianWest1_green := FALSE;
       "DB_ProcessData".crossroad_output.pedestrianWest1_red := FALSE;
       "DB_ProcessData".crossroad_output.pedestrianWest2_green := FALSE;
       "DB_ProcessData".crossroad_output.pedestrianWest2_red := FALSE;
       "DB_ProcessData".crossroad_output.trafficLightEast_green := FALSE;
       "DB_ProcessData".crossroad_output.trafficLightEast_red := FALSE;
       "DB_ProcessData".crossroad_output.trafficLightEast_yellow := FALSE;
       "DB_ProcessData".crossroad_output.trafficLightWest_green := FALSE;
       "DB_ProcessData".crossroad_output.trafficLightWest_red := FALSE;
       "DB_ProcessData".crossroad_output.trafficLightWest_yellow := FALSE;
       "DB_ProcessData".crossroad_output.trafficLightNorth_green := FALSE;
       "DB_ProcessData".crossroad_output.trafficLightNorth_red := FALSE;
       "DB_ProcessData".crossroad_output.trafficLightNorth_yellow := FALSE;
       "DB_ProcessData".crossroad_output.trafficLightSouth_green := FALSE;
       "DB_ProcessData".crossroad_output.trafficLightSouth_red := FALSE;
       "DB_ProcessData".crossroad_output.trafficLightSouth_yellow := FALSE;
   END_IF;
END_REGION

REGION Network 2: Night mode
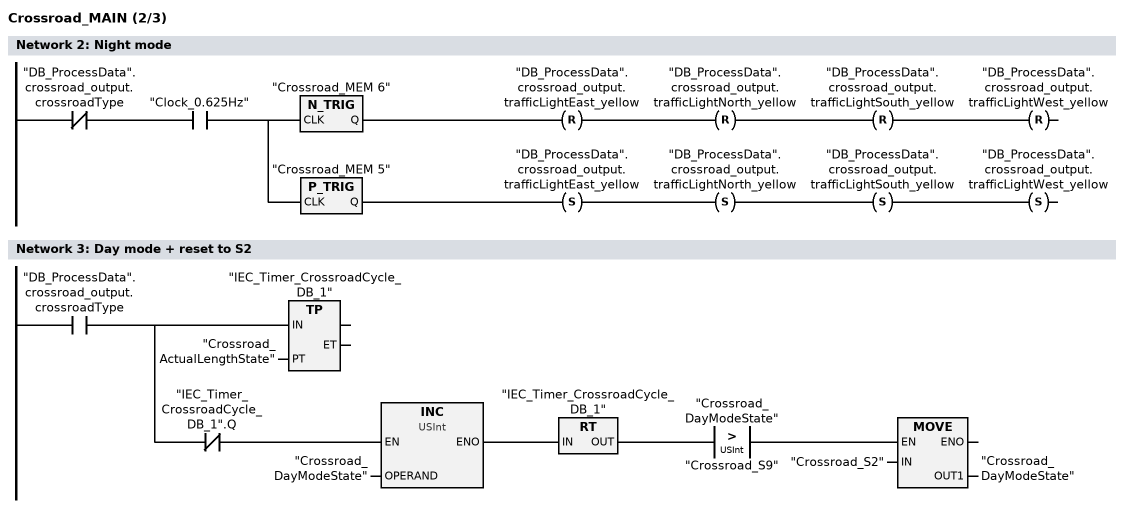
   RUNG wire#powerrail
      I_Contact( "DB_ProcessData".crossroad_output.crossroadType )
      Contact( "Clock_0.625Hz" )
      wire#w1
      N_Trig( "Crossroad_MEM 6" )
      R_Coil( "DB_ProcessData".crossroad_output.trafficLightEast_yellow )
      R_Coil( "DB_ProcessData".crossroad_output.trafficLightNorth_yellow )
      R_Coil( "DB_ProcessData".crossroad_output.trafficLightSouth_yellow )
      R_Coil( "DB_ProcessData".crossroad_output.trafficLightWest_yellow )
   END_RUNG
   RUNG wire#w1
      P_Trig( "Crossroad_MEM 5" )
      S_Coil( "DB_ProcessData".crossroad_output.trafficLightEast_yellow )
      S_Coil( "DB_ProcessData".crossroad_output.trafficLightNorth_yellow )
      S_Coil( "DB_ProcessData".crossroad_output.trafficLightSouth_yellow )
      S_Coil( "DB_ProcessData".crossroad_output.trafficLightWest_yellow )
   END_RUNG
   // the same network as SCL:
   #_w1 := NOT "DB_ProcessData".crossroad_output.crossroadType AND "Clock_0.625Hz";
   #_w2 := NOT #_w1 AND "Crossroad_MEM 6";   // falling edge
   "Crossroad_MEM 6" := #_w1;
   IF #_w2 THEN
       "DB_ProcessData".crossroad_output.trafficLightEast_yellow := FALSE;
       "DB_ProcessData".crossroad_output.trafficLightNorth_yellow := FALSE;
       "DB_ProcessData".crossroad_output.trafficLightSouth_yellow := FALSE;
       "DB_ProcessData".crossroad_output.trafficLightWest_yellow := FALSE;
   END_IF;
   #_w3 := #_w1 AND NOT "Crossroad_MEM 5";   // rising edge
   "Crossroad_MEM 5" := #_w1;
   IF #_w3 THEN
       "DB_ProcessData".crossroad_output.trafficLightEast_yellow := TRUE;
       "DB_ProcessData".crossroad_output.trafficLightNorth_yellow := TRUE;
       "DB_ProcessData".crossroad_output.trafficLightSouth_yellow := TRUE;
       "DB_ProcessData".crossroad_output.trafficLightWest_yellow := TRUE;
   END_IF;
END_REGION

REGION Network 3: Day mode + reset to S2
   "IEC_Timer_CrossroadCycle_DB_1".TP(IN := "DB_ProcessData".crossroad_output.crossroadType,
                           PT := "Crossroad_ActualLengthState");
   #_w1 := "DB_ProcessData".crossroad_output.crossroadType AND NOT "IEC_Timer_CrossroadCycle_DB_1".Q;
   IF #_w1 THEN
       "Crossroad_DayModeState" := "Crossroad_DayModeState" + 1;
       RESET_TIMER("IEC_Timer_CrossroadCycle_DB_1");
   END_IF;
   IF #_w1 AND ("Crossroad_DayModeState" > "Crossroad_S9") THEN
       "Crossroad_DayModeState" := "Crossroad_S2";
   END_IF;
END_REGION

REGION Network 4: Day mode time seq
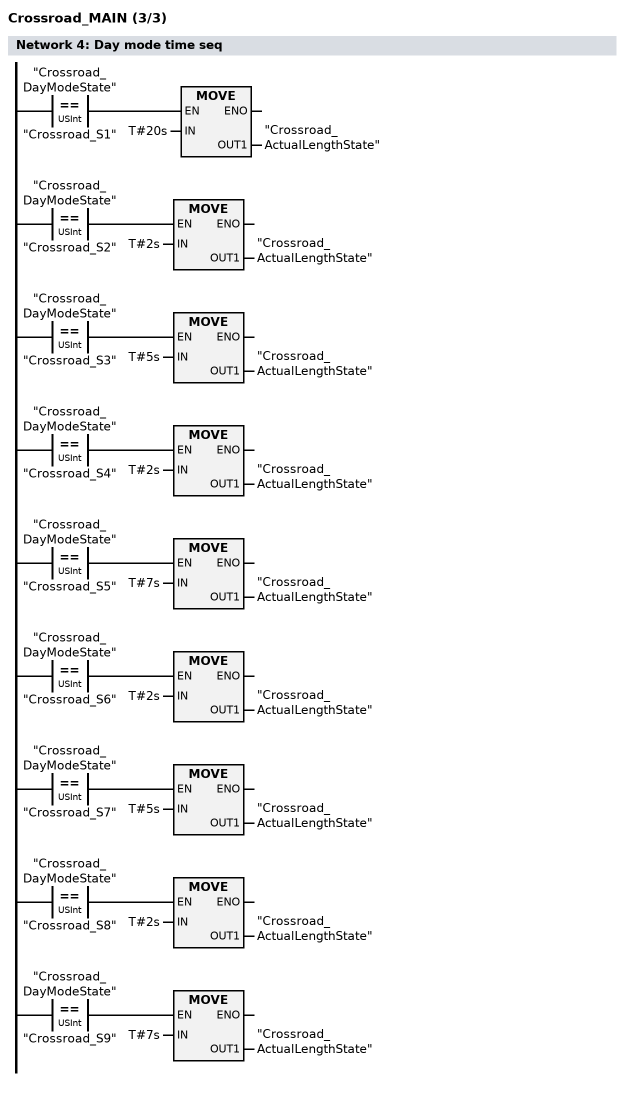
   RUNG wire#powerrail
      { S7_Templates := "SrcType := USInt" } EQ_Contact(in1 := "Crossroad_DayModeState", in2 := "Crossroad_S1")
      Move(in := T#20s, out1 => "Crossroad_ActualLengthState")
   END_RUNG
   RUNG wire#powerrail
      { S7_Templates := "SrcType := USInt" } EQ_Contact(in1 := "Crossroad_DayModeState", in2 := "Crossroad_S2")
      Move(in := T#2s, out1 => "Crossroad_ActualLengthState")
   END_RUNG
   RUNG wire#powerrail
      { S7_Templates := "SrcType := USInt" } EQ_Contact(in1 := "Crossroad_DayModeState", in2 := "Crossroad_S3")
      Move(in := T#5s, out1 => "Crossroad_ActualLengthState")
   END_RUNG
   RUNG wire#powerrail
      { S7_Templates := "SrcType := USInt" } EQ_Contact(in1 := "Crossroad_DayModeState", in2 := "Crossroad_S4")
      Move(in := T#2s, out1 => "Crossroad_ActualLengthState")
   END_RUNG
   RUNG wire#powerrail
      { S7_Templates := "SrcType := USInt" } EQ_Contact(in1 := "Crossroad_DayModeState", in2 := "Crossroad_S5")
      Move(in := T#7s, out1 => "Crossroad_ActualLengthState")
   END_RUNG
   RUNG wire#powerrail
      { S7_Templates := "SrcType := USInt" } EQ_Contact(in1 := "Crossroad_DayModeState", in2 := "Crossroad_S6")
      Move(in := T#2s, out1 => "Crossroad_ActualLengthState")
   END_RUNG
   RUNG wire#powerrail
      { S7_Templates := "SrcType := USInt" } EQ_Contact(in1 := "Crossroad_DayModeState", in2 := "Crossroad_S7")
      Move(in := T#5s, out1 => "Crossroad_ActualLengthState")
   END_RUNG
   RUNG wire#powerrail
      { S7_Templates := "SrcType := USInt" } EQ_Contact(in1 := "Crossroad_DayModeState", in2 := "Crossroad_S8")
      Move(in := T#2s, out1 => "Crossroad_ActualLengthState")
   END_RUNG
   RUNG wire#powerrail
      { S7_Templates := "SrcType := USInt" } EQ_Contact(in1 := "Crossroad_DayModeState", in2 := "Crossroad_S9")
      Move(in := T#7s, out1 => "Crossroad_ActualLengthState")
   END_RUNG
   // the same network as SCL:
   IF "Crossroad_DayModeState" = "Crossroad_S1" THEN "Crossroad_ActualLengthState" := T#20s; END_IF;
   IF "Crossroad_DayModeState" = "Crossroad_S2" THEN "Crossroad_ActualLengthState" := T#2s; END_IF;
   IF "Crossroad_DayModeState" = "Crossroad_S3" THEN "Crossroad_ActualLengthState" := T#5s; END_IF;
   IF "Crossroad_DayModeState" = "Crossroad_S4" THEN "Crossroad_ActualLengthState" := T#2s; END_IF;
   IF "Crossroad_DayModeState" = "Crossroad_S5" THEN "Crossroad_ActualLengthState" := T#7s; END_IF;
   IF "Crossroad_DayModeState" = "Crossroad_S6" THEN "Crossroad_ActualLengthState" := T#2s; END_IF;
   IF "Crossroad_DayModeState" = "Crossroad_S7" THEN "Crossroad_ActualLengthState" := T#5s; END_IF;
   IF "Crossroad_DayModeState" = "Crossroad_S8" THEN "Crossroad_ActualLengthState" := T#2s; END_IF;
   IF "Crossroad_DayModeState" = "Crossroad_S9" THEN "Crossroad_ActualLengthState" := T#7s; END_IF;
END_REGION

REGION Network 5 (SCL): Day mode lights
   IF "DB_ProcessData".crossroad_output.crossroadType THEN
       CASE "Crossroad_DayModeState" OF
           0:  // Statement section case S1
               // GREEN = FALSE, YELLOW = FALSE, RED = TRUE
               // PED: RED = TRUE, GREEN = FALSE

               "DB_ProcessData".crossroad_output.trafficLightEast_green := FALSE;
               "DB_ProcessData".crossroad_output.trafficLightEast_red := TRUE;
               "DB_ProcessData".crossroad_output.trafficLightEast_yellow := FALSE;

               "DB_ProcessData".crossroad_output.trafficLightNorth_green := FALSE;
               "DB_ProcessData".crossroad_output.trafficLightNorth_red := TRUE;
               "DB_ProcessData".crossroad_output.trafficLightNorth_yellow := FALSE;

               "DB_ProcessData".crossroad_output.trafficLightSouth_green := FALSE;
               "DB_ProcessData".crossroad_output.trafficLightSouth_red := TRUE;
               "DB_ProcessData".crossroad_output.trafficLightSouth_yellow := FALSE;

               "DB_ProcessData".crossroad_output.trafficLightWest_green := FALSE;
               "DB_ProcessData".crossroad_output.trafficLightWest_red := TRUE;
               "DB_ProcessData".crossroad_output.trafficLightWest_yellow := FALSE;

               "DB_ProcessData".crossroad_output.pedestrianSouth1_green := FALSE;
               "DB_ProcessData".crossroad_output.pedestrianSouth1_red := TRUE;
               "DB_ProcessData".crossroad_output.pedestrianSouth2_green := FALSE;
               "DB_ProcessData".crossroad_output.pedestrianSouth2_red := TRUE;

               "DB_ProcessData".crossroad_output.pedestrianWest1_green := FALSE;
               "DB_ProcessData".crossroad_output.pedestrianWest1_red := TRUE;
               "DB_ProcessData".crossroad_output.pedestrianWest2_green := FALSE;
               "DB_ProcessData".crossroad_output.pedestrianWest2_red := TRUE;

               //"PLC_LED_GREEN_1" := FALSE;
               //"PLC_LED_GREEN_2" := FALSE;
               //"PLC_LED_ORANGE_1" := FALSE;
               //"PLC_LED_ORANGE_2" := FALSE;
               //"PLC_LED_GREEN_CH" := FALSE;
               //"PLC_LED_RED_1" := TRUE;
               //"PLC_LED_RED_2" := TRUE;
               //"PLC_LED_RED_CH" := TRUE;

           1:  // Statement section case S2
               // GREEN = FALSE, RED = TRUE, YELLOW = TRUE
               // PED: RED = TRUE, GREEN = FALSE

               "DB_ProcessData".crossroad_output.trafficLightEast_green := FALSE;
               "DB_ProcessData".crossroad_output.trafficLightEast_red := TRUE;
               "DB_ProcessData".crossroad_output.trafficLightEast_yellow := TRUE;

               "DB_ProcessData".crossroad_output.trafficLightNorth_green := FALSE;
               "DB_ProcessData".crossroad_output.trafficLightNorth_red := TRUE;
               "DB_ProcessData".crossroad_output.trafficLightNorth_yellow := FALSE;

               "DB_ProcessData".crossroad_output.trafficLightSouth_green := FALSE;
               "DB_ProcessData".crossroad_output.trafficLightSouth_red := TRUE;
               "DB_ProcessData".crossroad_output.trafficLightSouth_yellow := FALSE;

               "DB_ProcessData".crossroad_output.trafficLightWest_green := FALSE;
               "DB_ProcessData".crossroad_output.trafficLightWest_red := TRUE;
               "DB_ProcessData".crossroad_output.trafficLightWest_yellow := TRUE;

               "DB_ProcessData".crossroad_output.pedestrianSouth1_green := FALSE;
               "DB_ProcessData".crossroad_output.pedestrianSouth1_red := TRUE;
               "DB_ProcessData".crossroad_output.pedestrianSouth2_green := FALSE;
               "DB_ProcessData".crossroad_output.pedestrianSouth2_red := TRUE;

               "DB_ProcessData".crossroad_output.pedestrianWest1_green := FALSE;
               "DB_ProcessData".crossroad_output.pedestrianWest1_red := TRUE;
               "DB_ProcessData".crossroad_output.pedestrianWest2_green := FALSE;
               "DB_ProcessData".crossroad_output.pedestrianWest2_red := TRUE;

               //"PLC_LED_GREEN_1" := FALSE;
               //"PLC_LED_GREEN_2" := FALSE;
               //"PLC_LED_ORANGE_1" := TRUE;
               //"PLC_LED_ORANGE_2" := FALSE;
               //"PLC_LED_GREEN_CH" := FALSE;
               //"PLC_LED_RED_1" := TRUE;
               //"PLC_LED_RED_2" := TRUE;
               //"PLC_LED_RED_CH" := TRUE;

           2:  // Statement section case S3
               // GREEN = TRUE, RED = FALSE, YELLOW = FALSE   // směr 1 (East, West)
               // GREEN = FALSE, RED = TRUE, YELLOW = FALSE   // směr 2 (North, South)
               // PED: RED = TRUE, GREEN = FALSE

               "DB_ProcessData".crossroad_output.trafficLightEast_green := TRUE;
               "DB_ProcessData".crossroad_output.trafficLightEast_red := FALSE;
               "DB_ProcessData".crossroad_output.trafficLightEast_yellow := FALSE;

               "DB_ProcessData".crossroad_output.trafficLightNorth_green := FALSE;
               "DB_ProcessData".crossroad_output.trafficLightNorth_red := TRUE;
               "DB_ProcessData".crossroad_output.trafficLightNorth_yellow := FALSE;

               "DB_ProcessData".crossroad_output.trafficLightSouth_green := FALSE;
               "DB_ProcessData".crossroad_output.trafficLightSouth_red := TRUE;
               "DB_ProcessData".crossroad_output.trafficLightSouth_yellow := FALSE;

               "DB_ProcessData".crossroad_output.trafficLightWest_green := TRUE;
               "DB_ProcessData".crossroad_output.trafficLightWest_red := FALSE;
               "DB_ProcessData".crossroad_output.trafficLightWest_yellow := FALSE;

               "DB_ProcessData".crossroad_output.pedestrianSouth1_green := FALSE;
               "DB_ProcessData".crossroad_output.pedestrianSouth1_red := TRUE;
               "DB_ProcessData".crossroad_output.pedestrianSouth2_green := FALSE;
               "DB_ProcessData".crossroad_output.pedestrianSouth2_red := TRUE;

               "DB_ProcessData".crossroad_output.pedestrianWest1_green := FALSE;
               "DB_ProcessData".crossroad_output.pedestrianWest1_red := TRUE;
               "DB_ProcessData".crossroad_output.pedestrianWest2_green := FALSE;
               "DB_ProcessData".crossroad_output.pedestrianWest2_red := TRUE;

               //"PLC_LED_GREEN_1" := TRUE;
               //"PLC_LED_GREEN_2" := FALSE;
               //"PLC_LED_ORANGE_1" := FALSE;
               //"PLC_LED_ORANGE_2" := FALSE;
               //"PLC_LED_GREEN_CH" := FALSE;
               //"PLC_LED_RED_1" := FALSE;
               //"PLC_LED_RED_2" := TRUE;
               //"PLC_LED_RED_CH" := TRUE;

           3:  // Statement section case S4
               // GREEN = FALSE, RED = FALSE, YELLOW = TRUE   // směr 1 (East, West)
               // GREEN = FALSE, RED = TRUE, YELLOW = FALSE   // směr 2 (North, South)
               // PED: RED = TRUE, GREEN = FALSE

               "DB_ProcessData".crossroad_output.trafficLightEast_green := FALSE;
               "DB_ProcessData".crossroad_output.trafficLightEast_red := FALSE;
               "DB_ProcessData".crossroad_output.trafficLightEast_yellow := TRUE;

               "DB_ProcessData".crossroad_output.trafficLightNorth_green := FALSE;
               "DB_ProcessData".crossroad_output.trafficLightNorth_red := TRUE;
               "DB_ProcessData".crossroad_output.trafficLightNorth_yellow := FALSE;

               "DB_ProcessData".crossroad_output.trafficLightSouth_green := FALSE;
               "DB_ProcessData".crossroad_output.trafficLightSouth_red := TRUE;
               "DB_ProcessData".crossroad_output.trafficLightSouth_yellow := FALSE;

               "DB_ProcessData".crossroad_output.trafficLightWest_green := FALSE;
               "DB_ProcessData".crossroad_output.trafficLightWest_red := FALSE;
               "DB_ProcessData".crossroad_output.trafficLightWest_yellow := TRUE;

               "DB_ProcessData".crossroad_output.pedestrianSouth1_green := FALSE;
               "DB_ProcessData".crossroad_output.pedestrianSouth1_red := TRUE;
               "DB_ProcessData".crossroad_output.pedestrianSouth2_green := FALSE;
               "DB_ProcessData".crossroad_output.pedestrianSouth2_red := TRUE;

               "DB_ProcessData".crossroad_output.pedestrianWest1_green := FALSE;
               "DB_ProcessData".crossroad_output.pedestrianWest1_red := TRUE;
               "DB_ProcessData".crossroad_output.pedestrianWest2_green := FALSE;
               "DB_ProcessData".crossroad_output.pedestrianWest2_red := TRUE;

               //"PLC_LED_GREEN_1" := FALSE;
               //"PLC_LED_GREEN_2" := FALSE;
               //"PLC_LED_ORANGE_1" := TRUE;
               //"PLC_LED_ORANGE_2" := FALSE;
               //"PLC_LED_GREEN_CH" := FALSE;
               //"PLC_LED_RED_1" := FALSE;
               //"PLC_LED_RED_2" := TRUE;
               //"PLC_LED_RED_CH" := TRUE;

           4:  // Statement section case S5
               // GREEN = FALSE, YELLOW = FALSE, RED = TRUE
               // PED: RED = TRUE, GREEN = FALSE

               "DB_ProcessData".crossroad_output.trafficLightEast_green := FALSE;
               "DB_ProcessData".crossroad_output.trafficLightEast_red := TRUE;
               "DB_ProcessData".crossroad_output.trafficLightEast_yellow := FALSE;

               "DB_ProcessData".crossroad_output.trafficLightNorth_green := FALSE;
               "DB_ProcessData".crossroad_output.trafficLightNorth_red := TRUE;
               "DB_ProcessData".crossroad_output.trafficLightNorth_yellow := FALSE;

               "DB_ProcessData".crossroad_output.trafficLightSouth_green := FALSE;
               "DB_ProcessData".crossroad_output.trafficLightSouth_red := TRUE;
               "DB_ProcessData".crossroad_output.trafficLightSouth_yellow := FALSE;

               "DB_ProcessData".crossroad_output.trafficLightWest_green := FALSE;
               "DB_ProcessData".crossroad_output.trafficLightWest_red := TRUE;
               "DB_ProcessData".crossroad_output.trafficLightWest_yellow := FALSE;

               "DB_ProcessData".crossroad_output.pedestrianSouth1_green := FALSE;
               "DB_ProcessData".crossroad_output.pedestrianSouth1_red := TRUE;
               "DB_ProcessData".crossroad_output.pedestrianSouth2_green := FALSE;
               "DB_ProcessData".crossroad_output.pedestrianSouth2_red := TRUE;

               "DB_ProcessData".crossroad_output.pedestrianWest1_green := FALSE;
               "DB_ProcessData".crossroad_output.pedestrianWest1_red := TRUE;
               "DB_ProcessData".crossroad_output.pedestrianWest2_green := FALSE;
               "DB_ProcessData".crossroad_output.pedestrianWest2_red := TRUE;

               //"PLC_LED_GREEN_1" := FALSE;
               //"PLC_LED_GREEN_2" := FALSE;
               //"PLC_LED_ORANGE_1" := FALSE;
               //"PLC_LED_ORANGE_2" := FALSE;
               //"PLC_LED_GREEN_CH" := FALSE;
               //"PLC_LED_RED_1" := TRUE;
               //"PLC_LED_RED_2" := TRUE;
               //"PLC_LED_RED_CH" := TRUE;

           5:  // Statement section case S6
               // GREEN = FALSE, RED = TRUE, YELLOW = FALSE   // směr 1 (East, West)
               // GREEN = FALSE, RED = TRUE, YELLOW = TRUE    // směr 2 (North, South)
               // PED: RED = TRUE, GREEN = FALSE (pokud není Crossroad_Walk_EN)

               "DB_ProcessData".crossroad_output.trafficLightEast_green := FALSE;
               "DB_ProcessData".crossroad_output.trafficLightEast_red := TRUE;
               "DB_ProcessData".crossroad_output.trafficLightEast_yellow := FALSE;

               "DB_ProcessData".crossroad_output.trafficLightNorth_green := FALSE;
               "DB_ProcessData".crossroad_output.trafficLightNorth_red := TRUE;
               "DB_ProcessData".crossroad_output.trafficLightNorth_yellow := TRUE;

               "DB_ProcessData".crossroad_output.trafficLightSouth_green := FALSE;
               "DB_ProcessData".crossroad_output.trafficLightSouth_red := TRUE;
               "DB_ProcessData".crossroad_output.trafficLightSouth_yellow := TRUE;

               "DB_ProcessData".crossroad_output.trafficLightWest_green := FALSE;
               "DB_ProcessData".crossroad_output.trafficLightWest_red := TRUE;
               "DB_ProcessData".crossroad_output.trafficLightWest_yellow := FALSE;

               "DB_ProcessData".crossroad_output.pedestrianSouth1_green := FALSE;
               "DB_ProcessData".crossroad_output.pedestrianSouth1_red := TRUE;
               "DB_ProcessData".crossroad_output.pedestrianSouth2_green := FALSE;
               "DB_ProcessData".crossroad_output.pedestrianSouth2_red := TRUE;

               "DB_ProcessData".crossroad_output.pedestrianWest1_green := FALSE;
               "DB_ProcessData".crossroad_output.pedestrianWest1_red := TRUE;
               "DB_ProcessData".crossroad_output.pedestrianWest2_green := FALSE;
               "DB_ProcessData".crossroad_output.pedestrianWest2_red := TRUE;

               //"PLC_LED_GREEN_1" := FALSE;
               //"PLC_LED_GREEN_2" := FALSE;
               //"PLC_LED_ORANGE_1" := FALSE;
               //"PLC_LED_ORANGE_2" := TRUE;
               //"PLC_LED_GREEN_CH" := FALSE;
               //"PLC_LED_RED_1" := TRUE;
               //"PLC_LED_RED_2" := TRUE;

               //"PLC_LED_GREEN_CH" := FALSE;
               //"PLC_LED_RED_CH" := TRUE;

               IF "Crossroad_Walk_EN" THEN
                   "DB_ProcessData".crossroad_output.pedestrianSouth1_green := TRUE;
                   "DB_ProcessData".crossroad_output.pedestrianSouth1_red := FALSE;
                   "DB_ProcessData".crossroad_output.pedestrianSouth2_green := TRUE;
                   "DB_ProcessData".crossroad_output.pedestrianSouth2_red := FALSE;

                   "DB_ProcessData".crossroad_output.pedestrianWest1_green := TRUE;
                   "DB_ProcessData".crossroad_output.pedestrianWest1_red := FALSE;
                   "DB_ProcessData".crossroad_output.pedestrianWest2_green := TRUE;
                   "DB_ProcessData".crossroad_output.pedestrianWest2_red := FALSE;

                   //"PLC_LED_GREEN_CH" := TRUE;
                   //"PLC_LED_RED_CH" := FALSE;
               END_IF;

           6:  // Statement section case S7
               // GREEN = FALSE, RED = TRUE, YELLOW = FALSE   // směr 1 (East, West)
               // GREEN = TRUE, RED = FALSE, YELLOW = FALSE   // směr 2 (North, South)
               // PED: RED = TRUE, GREEN = FALSE (pokud není Crossroad_Walk_EN)

               "DB_ProcessData".crossroad_output.trafficLightEast_green := FALSE;
               "DB_ProcessData".crossroad_output.trafficLightEast_red := TRUE;
               "DB_ProcessData".crossroad_output.trafficLightEast_yellow := FALSE;

               "DB_ProcessData".crossroad_output.trafficLightNorth_green := TRUE;
               "DB_ProcessData".crossroad_output.trafficLightNorth_red := FALSE;
               "DB_ProcessData".crossroad_output.trafficLightNorth_yellow := FALSE;

               "DB_ProcessData".crossroad_output.trafficLightSouth_green := TRUE;
               "DB_ProcessData".crossroad_output.trafficLightSouth_red := FALSE;
               "DB_ProcessData".crossroad_output.trafficLightSouth_yellow := FALSE;

               "DB_ProcessData".crossroad_output.trafficLightWest_green := FALSE;
               "DB_ProcessData".crossroad_output.trafficLightWest_red := TRUE;
               "DB_ProcessData".crossroad_output.trafficLightWest_yellow := FALSE;

               "DB_ProcessData".crossroad_output.pedestrianSouth1_green := FALSE;
               "DB_ProcessData".crossroad_output.pedestrianSouth1_red := TRUE;
               "DB_ProcessData".crossroad_output.pedestrianSouth2_green := FALSE;
               "DB_ProcessData".crossroad_output.pedestrianSouth2_red := TRUE;

               "DB_ProcessData".crossroad_output.pedestrianWest1_green := FALSE;
               "DB_ProcessData".crossroad_output.pedestrianWest1_red := TRUE;
               "DB_ProcessData".crossroad_output.pedestrianWest2_green := FALSE;
               "DB_ProcessData".crossroad_output.pedestrianWest2_red := TRUE;

               //"PLC_LED_GREEN_1" := FALSE;
               //"PLC_LED_GREEN_2" := TRUE;
               //"PLC_LED_ORANGE_1" := FALSE;
               //"PLC_LED_ORANGE_2" := FALSE;
               //"PLC_LED_RED_1" := TRUE;
               //"PLC_LED_RED_2" := FALSE;

               //"PLC_LED_GREEN_CH" := FALSE;
               //"PLC_LED_RED_CH" := TRUE;

               IF "Crossroad_Walk_EN" THEN
                   "DB_ProcessData".crossroad_output.pedestrianSouth1_green := TRUE;
                   "DB_ProcessData".crossroad_output.pedestrianSouth1_red := FALSE;
                   "DB_ProcessData".crossroad_output.pedestrianSouth2_green := TRUE;
                   "DB_ProcessData".crossroad_output.pedestrianSouth2_red := FALSE;

                   "DB_ProcessData".crossroad_output.pedestrianWest1_green := TRUE;
                   "DB_ProcessData".crossroad_output.pedestrianWest1_red := FALSE;
                   "DB_ProcessData".crossroad_output.pedestrianWest2_green := TRUE;
                   "DB_ProcessData".crossroad_output.pedestrianWest2_red := FALSE;

                   //"PLC_LED_GREEN_CH" := TRUE;
                   //"PLC_LED_RED_CH" := FALSE;
               END_IF;

           7:  // Statement section case S8
               // GREEN = FALSE, RED = TRUE, YELLOW = FALSE   // směr 1 (East, West)
               // GREEN = FALSE, RED = FALSE, YELLOW = TRUE   // směr 2 (North, South)
               // PED: RED = TRUE, GREEN = FALSE

               "DB_ProcessData".crossroad_output.trafficLightEast_green := FALSE;
               "DB_ProcessData".crossroad_output.trafficLightEast_red := TRUE;
               "DB_ProcessData".crossroad_output.trafficLightEast_yellow := FALSE;

               "DB_ProcessData".crossroad_output.trafficLightNorth_green := FALSE;
               "DB_ProcessData".crossroad_output.trafficLightNorth_red := FALSE;
               "DB_ProcessData".crossroad_output.trafficLightNorth_yellow := TRUE;

               "DB_ProcessData".crossroad_output.trafficLightSouth_green := FALSE;
               "DB_ProcessData".crossroad_output.trafficLightSouth_red := FALSE;
               "DB_ProcessData".crossroad_output.trafficLightSouth_yellow := TRUE;

               "DB_ProcessData".crossroad_output.trafficLightWest_green := FALSE;
               "DB_ProcessData".crossroad_output.trafficLightWest_red := TRUE;
               "DB_ProcessData".crossroad_output.trafficLightWest_yellow := FALSE;

               "DB_ProcessData".crossroad_output.pedestrianSouth1_green := FALSE;
               "DB_ProcessData".crossroad_output.pedestrianSouth1_red := TRUE;
               "DB_ProcessData".crossroad_output.pedestrianSouth2_green := FALSE;
               "DB_ProcessData".crossroad_output.pedestrianSouth2_red := TRUE;

               "DB_ProcessData".crossroad_output.pedestrianWest1_green := FALSE;
               "DB_ProcessData".crossroad_output.pedestrianWest1_red := TRUE;
               "DB_ProcessData".crossroad_output.pedestrianWest2_green := FALSE;
               "DB_ProcessData".crossroad_output.pedestrianWest2_red := TRUE;

               //"PLC_LED_GREEN_1" := FALSE;
               //"PLC_LED_GREEN_2" := FALSE;
               //"PLC_LED_ORANGE_1" := FALSE;
               //"PLC_LED_ORANGE_2" := TRUE;
               //"PLC_LED_GREEN_CH" := FALSE;
               //"PLC_LED_RED_1" := TRUE;
               //"PLC_LED_RED_2" := FALSE;
               //"PLC_LED_RED_CH" := TRUE;

           8:  // Statement section case S9
               // GREEN = FALSE, YELLOW = FALSE, RED = TRUE
               // PED: RED = TRUE, GREEN = FALSE

               "DB_ProcessData".crossroad_output.trafficLightEast_green := FALSE;
               "DB_ProcessData".crossroad_output.trafficLightEast_red := TRUE;
               "DB_ProcessData".crossroad_output.trafficLightEast_yellow := FALSE;

               "DB_ProcessData".crossroad_output.trafficLightNorth_green := FALSE;
               "DB_ProcessData".crossroad_output.trafficLightNorth_red := TRUE;
               "DB_ProcessData".crossroad_output.trafficLightNorth_yellow := FALSE;

               "DB_ProcessData".crossroad_output.trafficLightSouth_green := FALSE;
               "DB_ProcessData".crossroad_output.trafficLightSouth_red := TRUE;
               "DB_ProcessData".crossroad_output.trafficLightSouth_yellow := FALSE;

               "DB_ProcessData".crossroad_output.trafficLightWest_green := FALSE;
               "DB_ProcessData".crossroad_output.trafficLightWest_red := TRUE;
               "DB_ProcessData".crossroad_output.trafficLightWest_yellow := FALSE;

               "DB_ProcessData".crossroad_output.pedestrianSouth1_green := FALSE;
               "DB_ProcessData".crossroad_output.pedestrianSouth1_red := TRUE;
               "DB_ProcessData".crossroad_output.pedestrianSouth2_green := FALSE;
               "DB_ProcessData".crossroad_output.pedestrianSouth2_red := TRUE;

               "DB_ProcessData".crossroad_output.pedestrianWest1_green := FALSE;
               "DB_ProcessData".crossroad_output.pedestrianWest1_red := TRUE;
               "DB_ProcessData".crossroad_output.pedestrianWest2_green := FALSE;
               "DB_ProcessData".crossroad_output.pedestrianWest2_red := TRUE;

               //"PLC_LED_GREEN_1" := FALSE;
               //"PLC_LED_GREEN_2" := FALSE;
               //"PLC_LED_ORANGE_1" := FALSE;
               //"PLC_LED_ORANGE_2" := FALSE;
               //"PLC_LED_GREEN_CH" := FALSE;
               //"PLC_LED_RED_1" := TRUE;
               //"PLC_LED_RED_2" := TRUE;
               //"PLC_LED_RED_CH" := TRUE;

               "Crossroad_Walk_EN" := FALSE;

           ELSE  // Statement section ELSE
               "DB_ProcessData".crossroad_output.trafficLightEast_green := FALSE;
               "DB_ProcessData".crossroad_output.trafficLightEast_red := FALSE;
               "DB_ProcessData".crossroad_output.trafficLightEast_yellow := FALSE;

               "DB_ProcessData".crossroad_output.trafficLightNorth_green := FALSE;
               "DB_ProcessData".crossroad_output.trafficLightNorth_red := FALSE;
               "DB_ProcessData".crossroad_output.trafficLightNorth_yellow := FALSE;

               "DB_ProcessData".crossroad_output.trafficLightSouth_green := FALSE;
               "DB_ProcessData".crossroad_output.trafficLightSouth_red := FALSE;
               "DB_ProcessData".crossroad_output.trafficLightSouth_yellow := FALSE;

               "DB_ProcessData".crossroad_output.trafficLightWest_green := FALSE;
               "DB_ProcessData".crossroad_output.trafficLightWest_red := FALSE;
               "DB_ProcessData".crossroad_output.trafficLightWest_yellow := FALSE;

               "DB_ProcessData".crossroad_output.pedestrianSouth1_green := FALSE;
               "DB_ProcessData".crossroad_output.pedestrianSouth1_red := FALSE;
               "DB_ProcessData".crossroad_output.pedestrianSouth2_green := FALSE;
               "DB_ProcessData".crossroad_output.pedestrianSouth2_red := FALSE;

               "DB_ProcessData".crossroad_output.pedestrianWest1_green := FALSE;
               "DB_ProcessData".crossroad_output.pedestrianWest1_red := FALSE;
               "DB_ProcessData".crossroad_output.pedestrianWest2_green := FALSE;
               "DB_ProcessData".crossroad_output.pedestrianWest2_red := FALSE;

               //"PLC_LED_GREEN_1" := FALSE;
               //"PLC_LED_GREEN_2" := FALSE;
               //"PLC_LED_ORANGE_1" := FALSE;
               //"PLC_LED_ORANGE_2" := FALSE;
               //"PLC_LED_RED_1" := FALSE;
               //"PLC_LED_RED_2" := FALSE;
               //"PLC_LED_GREEN_CH" := FALSE;
               //"PLC_LED_RED_CH" := FALSE;

               "Crossroad_Walk_EN" := FALSE;
       END_CASE;
   END_IF;
END_REGION

REGION Network 6 (SCL): Pedestrians bnts
   IF "DB_ProcessData".crossroad_input.btnSouthCrosswalk1 OR "DB_ProcessData".crossroad_input.btnSouthCrosswalk2 OR "DB_ProcessData".crossroad_input.btnWestCrosswalk1 OR "DB_ProcessData".crossroad_input.btnWestCrosswalk2 THEN
       "Crossroad_Walk_EN" := TRUE;
   END_IF;
END_REGION
END_FUNCTION

// folder: Crosswalk

FUNCTION "Crosswalk_MAIN" : Void   // FC1, LAD
{ S7_Optimized_Access := 'TRUE' }
VERSION : 0.1
BEGIN

REGION Network 1: Control
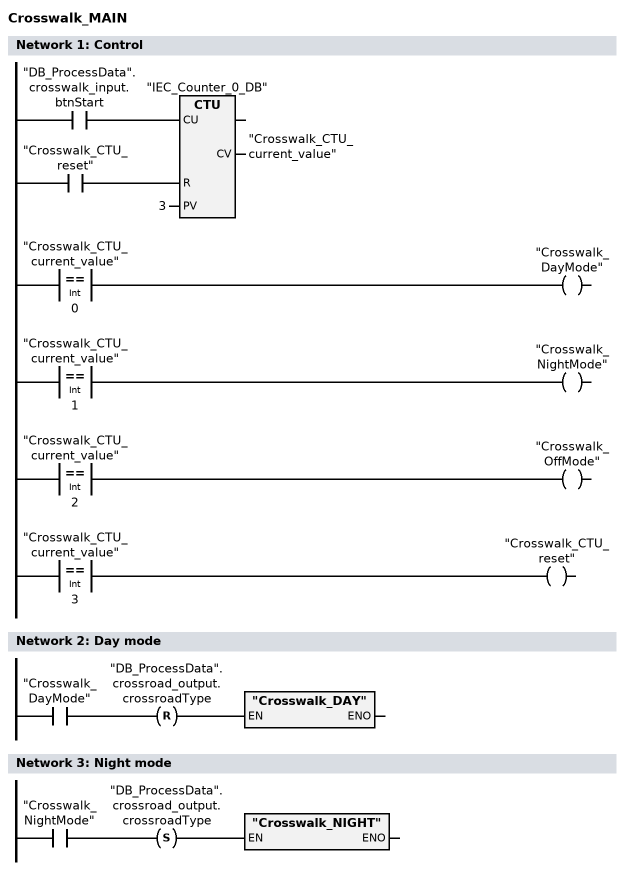
   "IEC_Counter_0_DB".CTU(CU := "DB_ProcessData".crosswalk_input.btnStart,
                          R := "Crosswalk_CTU_reset",
                          PV := 3,
                          CV => "Crosswalk_CTU_current_value");
   "Crosswalk_DayMode" := "Crosswalk_CTU_current_value" = 0;
   "Crosswalk_NightMode" := "Crosswalk_CTU_current_value" = 1;
   "Crosswalk_OffMode" := "Crosswalk_CTU_current_value" = 2;
   "Crosswalk_CTU_reset" := "Crosswalk_CTU_current_value" = 3;
END_REGION

REGION Network 2: Day mode
   RUNG wire#powerrail
      Contact( "Crosswalk_DayMode" )
      R_Coil( "DB_ProcessData".crossroad_output.crossroadType )
      "Crosswalk_DAY"()
   END_RUNG
   // the same network as SCL:
   IF "Crosswalk_DayMode" THEN
       "DB_ProcessData".crossroad_output.crossroadType := FALSE;
       "Crosswalk_DAY"();
   END_IF;
END_REGION

REGION Network 3: Night mode
   RUNG wire#powerrail
      Contact( "Crosswalk_NightMode" )
      S_Coil( "DB_ProcessData".crossroad_output.crossroadType )
      "Crosswalk_NIGHT"()
   END_RUNG
   // the same network as SCL:
   IF "Crosswalk_NightMode" THEN
       "DB_ProcessData".crossroad_output.crossroadType := TRUE;
       "Crosswalk_NIGHT"();
   END_IF;
END_REGION

REGION Network 4 (SCL): Off mode
   IF "Crosswalk_OffMode" = TRUE THEN
       "DB_ProcessData".crosswalk_output.pedestrianLightGreen1 := FALSE;
       "DB_ProcessData".crosswalk_output.pedestrianLightGreen2 := FALSE;
       "DB_ProcessData".crosswalk_output.pedestrianLightRed1 := FALSE;
       "DB_ProcessData".crosswalk_output.pedestrianLightRed2 := FALSE;
       "DB_ProcessData".crosswalk_output.trafficLightGreen1 := FALSE;
       "DB_ProcessData".crosswalk_output.trafficLightGreen2 := FALSE;
       "DB_ProcessData".crosswalk_output.trafficLightsRed1 := FALSE;
       "DB_ProcessData".crosswalk_output.trafficLightsRed2 := FALSE;
       "DB_ProcessData".crosswalk_output.trafficLightsYellow1 := FALSE;
       "DB_ProcessData".crosswalk_output.trafficLightsYellow2 := FALSE;
   END_IF;
END_REGION
END_FUNCTION

FUNCTION "Crosswalk_DAY" : Void   // FC2, LAD
{ S7_Optimized_Access := 'TRUE' }
VERSION : 0.1
   VAR_TEMP   // added for the SCL form of the ladder/FBD networks
      _w1 : Bool;
   END_VAR
BEGIN

REGION Network 1: Green
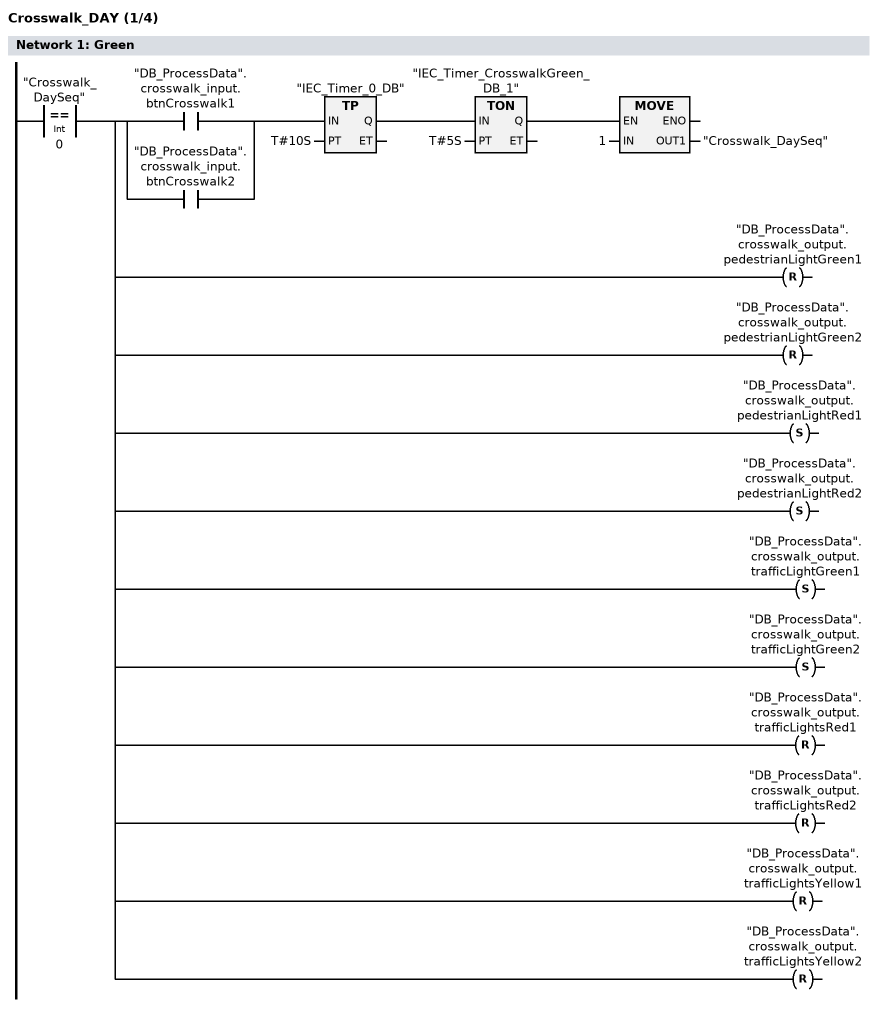
   #_w1 := "Crosswalk_DaySeq" = 0;
   "IEC_Timer_0_DB".TP(IN := #_w1 AND ("DB_ProcessData".crosswalk_input.btnCrosswalk1 OR "DB_ProcessData".crosswalk_input.btnCrosswalk2),
                       PT := T#10S);
   "IEC_Timer_CrosswalkGreen_DB_1".TON(IN := "IEC_Timer_0_DB".Q, PT := T#5S);
   IF "IEC_Timer_CrosswalkGreen_DB_1".Q THEN "Crosswalk_DaySeq" := 1; END_IF;
   IF #_w1 THEN
       "DB_ProcessData".crosswalk_output.pedestrianLightGreen1 := FALSE;
       "DB_ProcessData".crosswalk_output.pedestrianLightGreen2 := FALSE;
       "DB_ProcessData".crosswalk_output.pedestrianLightRed1 := TRUE;
       "DB_ProcessData".crosswalk_output.pedestrianLightRed2 := TRUE;
       "DB_ProcessData".crosswalk_output.trafficLightGreen1 := TRUE;
       "DB_ProcessData".crosswalk_output.trafficLightGreen2 := TRUE;
       "DB_ProcessData".crosswalk_output.trafficLightsRed1 := FALSE;
       "DB_ProcessData".crosswalk_output.trafficLightsRed2 := FALSE;
       "DB_ProcessData".crosswalk_output.trafficLightsYellow1 := FALSE;
       "DB_ProcessData".crosswalk_output.trafficLightsYellow2 := FALSE;
   END_IF;
END_REGION

REGION Network 2: Yellow1
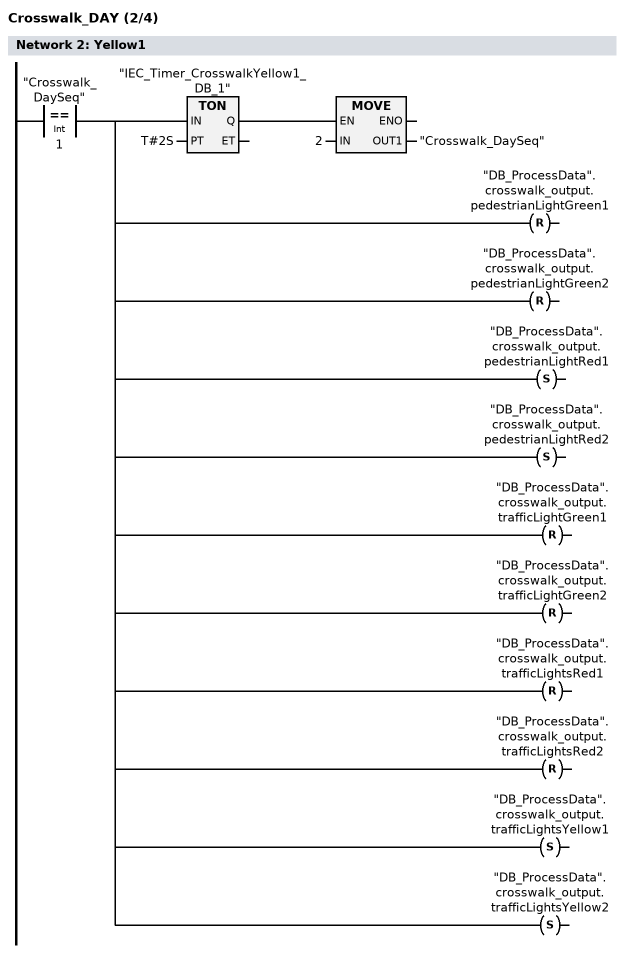
   #_w1 := "Crosswalk_DaySeq" = 1;
   "IEC_Timer_CrosswalkYellow1_DB_1".TON(IN := #_w1, PT := T#2S);
   IF "IEC_Timer_CrosswalkYellow1_DB_1".Q THEN "Crosswalk_DaySeq" := 2; END_IF;
   IF #_w1 THEN
       "DB_ProcessData".crosswalk_output.pedestrianLightGreen1 := FALSE;
       "DB_ProcessData".crosswalk_output.pedestrianLightGreen2 := FALSE;
       "DB_ProcessData".crosswalk_output.pedestrianLightRed1 := TRUE;
       "DB_ProcessData".crosswalk_output.pedestrianLightRed2 := TRUE;
       "DB_ProcessData".crosswalk_output.trafficLightGreen1 := FALSE;
       "DB_ProcessData".crosswalk_output.trafficLightGreen2 := FALSE;
       "DB_ProcessData".crosswalk_output.trafficLightsRed1 := FALSE;
       "DB_ProcessData".crosswalk_output.trafficLightsRed2 := FALSE;
       "DB_ProcessData".crosswalk_output.trafficLightsYellow1 := TRUE;
       "DB_ProcessData".crosswalk_output.trafficLightsYellow2 := TRUE;
   END_IF;
END_REGION

REGION Network 3: Red
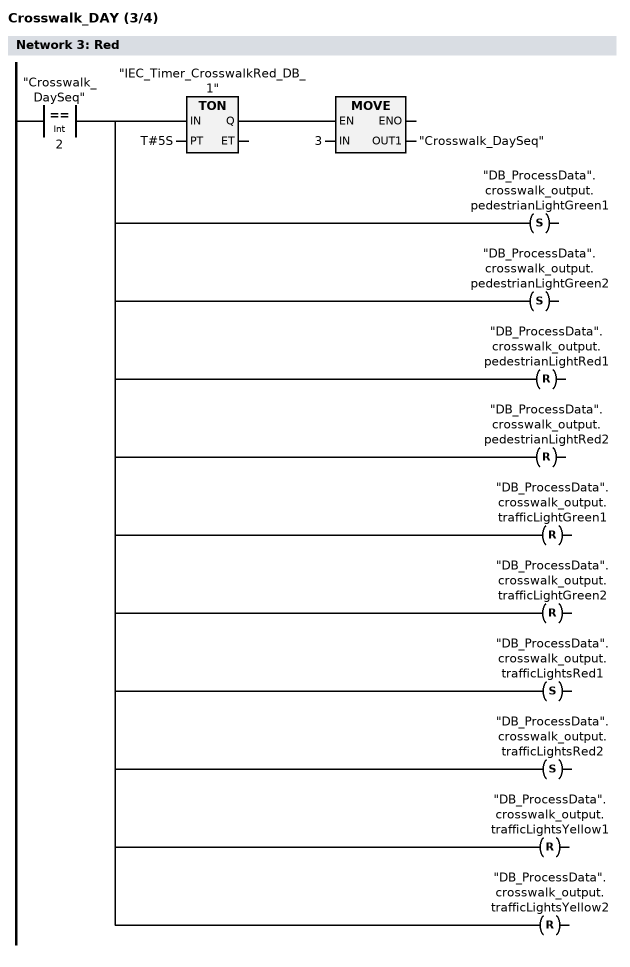
   #_w1 := "Crosswalk_DaySeq" = 2;
   "IEC_Timer_CrosswalkRed_DB_1".TON(IN := #_w1, PT := T#5S);
   IF "IEC_Timer_CrosswalkRed_DB_1".Q THEN "Crosswalk_DaySeq" := 3; END_IF;
   IF #_w1 THEN
       "DB_ProcessData".crosswalk_output.pedestrianLightGreen1 := TRUE;
       "DB_ProcessData".crosswalk_output.pedestrianLightGreen2 := TRUE;
       "DB_ProcessData".crosswalk_output.pedestrianLightRed1 := FALSE;
       "DB_ProcessData".crosswalk_output.pedestrianLightRed2 := FALSE;
       "DB_ProcessData".crosswalk_output.trafficLightGreen1 := FALSE;
       "DB_ProcessData".crosswalk_output.trafficLightGreen2 := FALSE;
       "DB_ProcessData".crosswalk_output.trafficLightsRed1 := TRUE;
       "DB_ProcessData".crosswalk_output.trafficLightsRed2 := TRUE;
       "DB_ProcessData".crosswalk_output.trafficLightsYellow1 := FALSE;
       "DB_ProcessData".crosswalk_output.trafficLightsYellow2 := FALSE;
   END_IF;
END_REGION

REGION Network 4: Yellow2
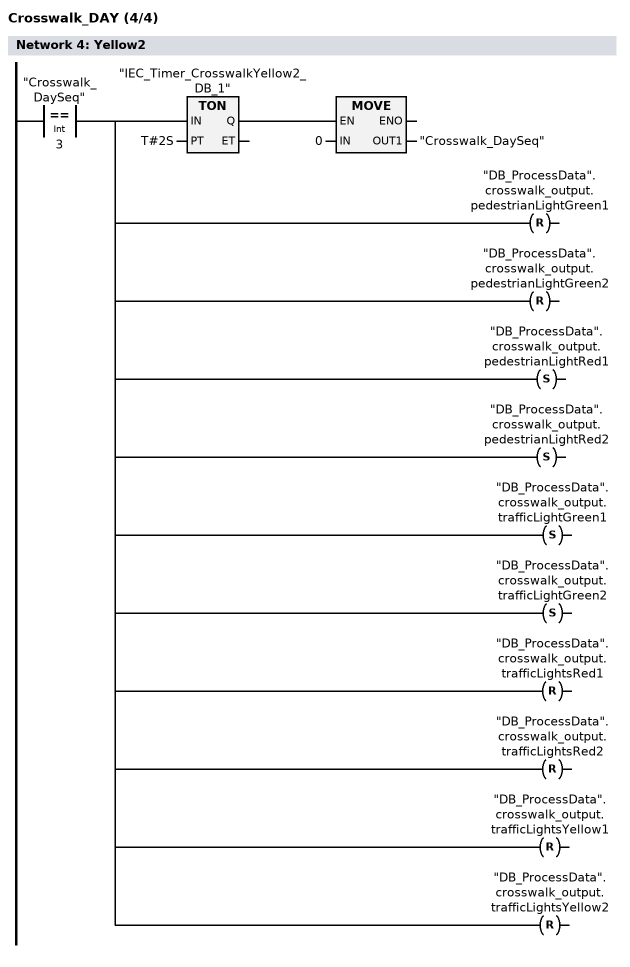
   #_w1 := "Crosswalk_DaySeq" = 3;
   "IEC_Timer_CrosswalkYellow2_DB_1".TON(IN := #_w1, PT := T#2S);
   IF "IEC_Timer_CrosswalkYellow2_DB_1".Q THEN "Crosswalk_DaySeq" := 0; END_IF;
   IF #_w1 THEN
       "DB_ProcessData".crosswalk_output.pedestrianLightGreen1 := FALSE;
       "DB_ProcessData".crosswalk_output.pedestrianLightGreen2 := FALSE;
       "DB_ProcessData".crosswalk_output.pedestrianLightRed1 := TRUE;
       "DB_ProcessData".crosswalk_output.pedestrianLightRed2 := TRUE;
       "DB_ProcessData".crosswalk_output.trafficLightGreen1 := TRUE;
       "DB_ProcessData".crosswalk_output.trafficLightGreen2 := TRUE;
       "DB_ProcessData".crosswalk_output.trafficLightsRed1 := FALSE;
       "DB_ProcessData".crosswalk_output.trafficLightsRed2 := FALSE;
       "DB_ProcessData".crosswalk_output.trafficLightsYellow1 := FALSE;
       "DB_ProcessData".crosswalk_output.trafficLightsYellow2 := FALSE;
   END_IF;
END_REGION
END_FUNCTION

FUNCTION "Crosswalk_NIGHT" : Void   // FC3, LAD
{ S7_Optimized_Access := 'TRUE' }
VERSION : 0.1
   VAR_TEMP   // added for the SCL form of the ladder/FBD networks
      _w1 : Bool;
   END_VAR
BEGIN

REGION Network 1: On
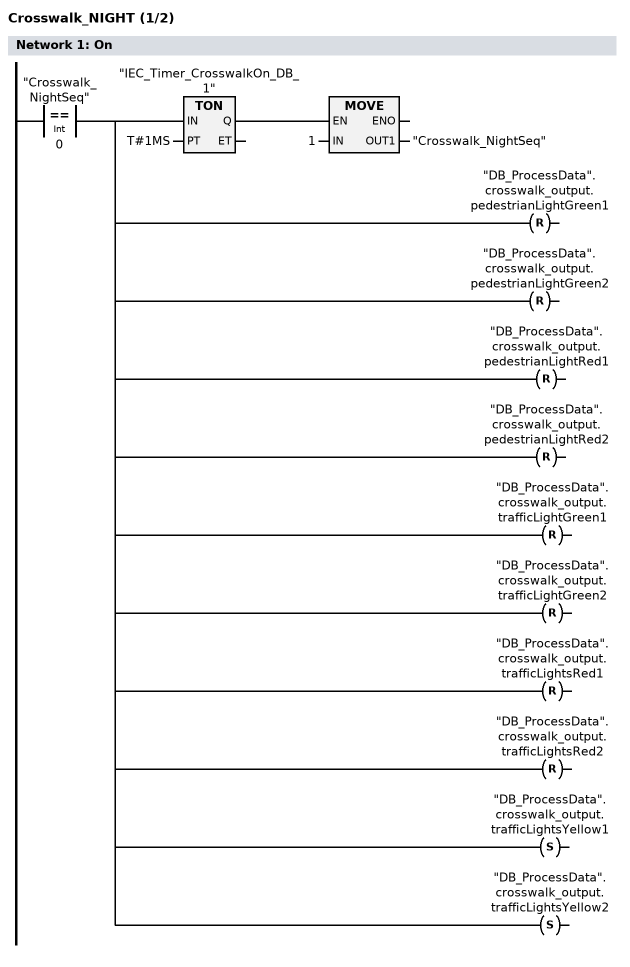
   #_w1 := "Crosswalk_NightSeq" = 0;
   "IEC_Timer_CrosswalkOn_DB_1".TON(IN := #_w1, PT := T#1MS);
   IF "IEC_Timer_CrosswalkOn_DB_1".Q THEN "Crosswalk_NightSeq" := 1; END_IF;
   IF #_w1 THEN
       "DB_ProcessData".crosswalk_output.pedestrianLightGreen1 := FALSE;
       "DB_ProcessData".crosswalk_output.pedestrianLightGreen2 := FALSE;
       "DB_ProcessData".crosswalk_output.pedestrianLightRed1 := FALSE;
       "DB_ProcessData".crosswalk_output.pedestrianLightRed2 := FALSE;
       "DB_ProcessData".crosswalk_output.trafficLightGreen1 := FALSE;
       "DB_ProcessData".crosswalk_output.trafficLightGreen2 := FALSE;
       "DB_ProcessData".crosswalk_output.trafficLightsRed1 := FALSE;
       "DB_ProcessData".crosswalk_output.trafficLightsRed2 := FALSE;
       "DB_ProcessData".crosswalk_output.trafficLightsYellow1 := TRUE;
       "DB_ProcessData".crosswalk_output.trafficLightsYellow2 := TRUE;
   END_IF;
END_REGION

REGION Network 2: Off
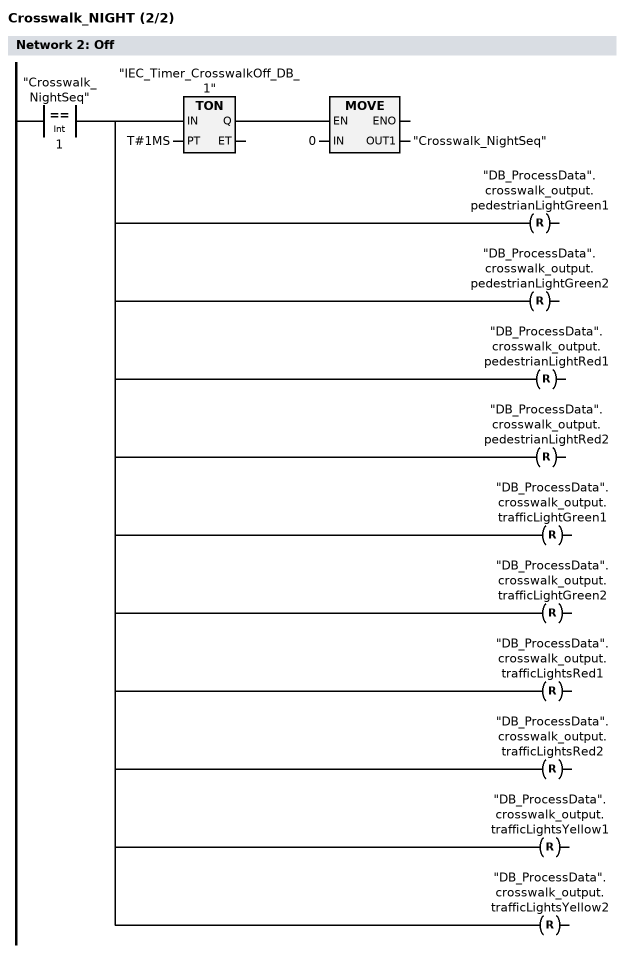
   #_w1 := "Crosswalk_NightSeq" = 1;
   "IEC_Timer_CrosswalkOff_DB_1".TON(IN := #_w1, PT := T#1MS);
   IF "IEC_Timer_CrosswalkOff_DB_1".Q THEN "Crosswalk_NightSeq" := 0; END_IF;
   IF #_w1 THEN
       "DB_ProcessData".crosswalk_output.pedestrianLightGreen1 := FALSE;
       "DB_ProcessData".crosswalk_output.pedestrianLightGreen2 := FALSE;
       "DB_ProcessData".crosswalk_output.pedestrianLightRed1 := FALSE;
       "DB_ProcessData".crosswalk_output.pedestrianLightRed2 := FALSE;
       "DB_ProcessData".crosswalk_output.trafficLightGreen1 := FALSE;
       "DB_ProcessData".crosswalk_output.trafficLightGreen2 := FALSE;
       "DB_ProcessData".crosswalk_output.trafficLightsRed1 := FALSE;
       "DB_ProcessData".crosswalk_output.trafficLightsRed2 := FALSE;
       "DB_ProcessData".crosswalk_output.trafficLightsYellow1 := FALSE;
       "DB_ProcessData".crosswalk_output.trafficLightsYellow2 := FALSE;
   END_IF;
END_REGION
END_FUNCTION

// folder: LHTTP

FUNCTION_BLOCK "LHTTP_Get"   // FB8, SCL
TITLE = LHTTP_Get
{ S7_Optimized_Access := 'TRUE' }
AUTHOR : Siemens Industry Online Support
FAMILY : LHTTP
VERSION : 2.2
// Implements the HTTP GET method
   VAR_INPUT
      execute : Bool;   // Send HTTP request
      hwID : Hw_Any;   // Hardware ID of Ethernet interface
      connID : Conn_Ouc := 1;   // Unique connection ID
      url : String;   // URL, i.e. "http://www.siemens.com/simatic"
      queryParams : String;   // Additional query parameters if "url" is not long enough, i.e. "lang=en&q=simatic"; "?" or "&" is inserted automatically in between "url" and "queryParameters". / Optional query parameters that are appended to URL, i.e. "lang=en&q=simatic"
      userFields : Array[0..#UPPER_USER_FIELDS] of Char;   // Additional user-defined header fields
      tls : "LHTTP_typeTLS";   // TLS certificates for secure connections (HTTPS), leave open for non-secure connections (HTTP)
      keepConnection : Bool;   // Keep connection established after execution of request
      timeOut : Time := T#10s;   // Time to wait for response from server
   END_VAR
   VAR_OUTPUT
      connected : Bool;   // Connection to web server is established
      done : Bool;   // HTTP request finished
      busy : Bool;   // Function is busy
      error : Bool;   // An error occured
      status : Word := 16#7000;   // Specifies the error
      diagnostics : "typeDiagnostics";   // Diagnostics information of FB
      responseCode : UInt;   // HTTP response code
      length : UDInt;   // Length of received data
   END_VAR
   VAR_IN_OUT
      responseData : Array[*] of Char;   // Data received from HTTP server
   END_VAR
   VAR
      instTSendC : TSEND_C;   // Instance of TSEND_C
      instTRcv : TRCV;   // Instance of TRCV
      instTimeout : TON_TIME;   // Time-out
      statConnected : Bool;   // Static value for output 'connected'
      statDone : Bool;   // Static value for output 'done'
      statBusy : Bool;   // Static value for output 'busy'
      statError : Bool;   // Static value for output 'error'
      statStatus : Word := 16#7000;   // Static value for output 'status'
      statResponseCode : UInt;   // Static value for output 'responseCode'
      statLength : UDInt;   // Static value for output 'length'
      statFBState : USInt := 0;   // Current state in state machine
      statSubfunctionStatus : DWord;   // Status or return value of called FBs, FCs and system blocks
      statEmptyDiagnostics : "typeDiagnostics";   // Empty diagnostics information (for initialization purposes only)
      statParam : Struct   // Connection parameters
         isQDN : Bool;
         paramQDN : TCON_QDN_SEC;   // Connection parameters in form of QDN
         paramIP : TCON_IP_V4_SEC;   // Connection parameters in form of IP address
      END_STRUCT;
      statHost : String;   // Host part of URL
      statRequest : Struct   // GET request
         chars : Array[0..#UPPER_REQUEST_ARRAY] of Char;   // GET request (max. length: url (254) + data (254) + header (94)
         length : UInt;   // Length of GET request
      END_STRUCT;
      statSend : Struct   // Parameters for instruction TSend_C
         connect : Bool;   // Establish and keep connection
         req : Bool;   // Send data
      END_STRUCT;
      statEncoding : String;   // Transfer encoding of response from HTTP server
      statContentLength : UDInt;   // Content length as specified in header of response
      statChunkLen : UDInt;   // Remaining length of current chunk
      statRcvdLen : UDInt;   // Sum length of received data
      statTimeoutIn : Bool;   // Timeout
      statRcvBuffer : Array[0..#UPPER_TCP_FRAME] of Char;   // Temporary receive buffer
      statSizeRcvArray : UDInt;   // Size of receive buffer at parameter "responseData"
      statExecuteOld : Bool;   // Last cycle's value of input "execute"
      statHeaderComplete : Bool;   // Header was received completely
   END_VAR
   VAR_TEMP
      tempUrl : String;   // Copy of URL
      tempQuery : String;   // Query part of URL
      tempIndex : DInt;   // Index for for loops
      tempPos : Int;   // General tag for positions
      tempLen : UInt;   // General tag for lengths
      tempRet : Word;   // General tag for return values
      tempString : String;   // General tag for strings
      tempExitLoop : Bool;   // Condition to exit REPEAT loop around state machine
      tempChunk : Struct   // Temporary tags for chunked encoding
         posData : UInt;   // Start position of data in current packet
         lenData : UInt;   // Length of data in current packet
         exitLoop : Bool;   // Condition to exit loop
      END_STRUCT;
   END_VAR
   VAR CONSTANT
      UPPER_REQUEST_ARRAY : UInt := 1459;   // Upper limit of request array
      UPPER_TCP_FRAME : UInt := 1459;   // Upper limit of a TCP/IP frame
      UPPER_USER_FIELDS : USInt := 255;   // Upper limit of userFields
      PORT_UNSECURE : UInt := 80;   // Port for unsecure HTTP connection
      PORT_SECURE : UInt := 443;   // Port for secure HTTP connection
      POS_RESPONSE_CODE : USInt := 9;   // Position of HTTP response code in response message
      STATUS_DONE : Word := 16#0000;   // Job finished without errors
      STATUS_DISCONNECTED : Word := 16#0003;   // Communication connection closed
      STATUS_IDLE : Word := 16#7000;   // No job
      STATUS_FIRST_CALL : Word := 16#7001;   // First call after incoming new job (rising edge 'execute')
      STATUS_CONNECTING : Word := 16#7002;   // Connection is currently being established
      STATUS_DISCONNECTING : Word := 16#7003;   // Communication connection is being terminated
      STATUS_MONITORING : Word := 16#7004;   // Communication connection has been established and is being monitored. No send job execution active
      STATUS_SENT : Word := 16#7005;   // Request sent, waiting for response
      SUB_STATUS_NO_ERROR : DWord := 16#0000_0000;   // No error occured in subfunction call
      ERR_BOUND_NOT_ZERO : Word := 16#8201;   // Lower bound of receive buffer is not 0
      ERR_INVALID_URL : Word := 16#8202;   // Invalid URL
      ERR_DIFFERENT_HOST : Word := 16#8203;   // Trying to use existing connection with different host
      ERR_END_USER_FIELDS : Word := 16#8206;   // End of user-defined header fields could not be found
      ERR_REQUEST_SIZE : Word := 16#8210;   // Request array is too small for specified parameters
      ERR_RESPONSE_SIZE : Word := 16#8220;   // Receive buffer at parameter "responseData" too small
      ERR_CONN_LOST : Word := 16#8400;   // Offset for lost connection
      ERR_FORWARDING : Word := 16#8403;   // Server responded with forwarding message. Forwarding is not supported, see "diagnostics"
      ERR_WEBSERVER : Word := 16#8404;   // Webserver responded with error code, see "diagnostics"
      ERR_INVALID_HEADER : Word := 16#8405;   // Header of response is invalid or incomplete / Header of response is invalid
      ERR_TIMEOUT : Word := 16#8408;   // Time-out occurred
      ERR_UNDEFINED_STATE : Word := 16#8600;   // Error due to an undefined state in state machine
      ERR_TSENDC : Word := 16#8601;   // Error: TCON encountered an error, see "diagnostics"
      ERR_TRCV : Word := 16#8603;   // Error: TURCV encountered error, see "diagnostics"
      ERR_MOVE_USER_FIELDS : Word := 16#8612;   // Error in MOVE_BLK_VARIANT to copy user-defined header fields, see "diagnostics"
      ERR_ENCODING_UNKNOWN : Word := 16#8620;   // Transfer encoding of response could not be detected or is unsupported
      ERR_MOVE_IDENTITY : Word := 16#8630;   // Error in MOVE_BLK_VARIANT for transfer encoding 'identity', see "diagnostics"
      ERR_DECODING_FAILED : Word := 16#8640;   // Chunk encoded response could not be decoded
      ERR_MOVE_CHUNKED : Word := 16#8641;   // Error in MOVE_BLK_VARIANT for transfer encoding 'chunked', see "diagnostics"
      TSENDC_STATUS_CONNECTED : Word := 16#0001;   // TSEND_C: Communication connection established
      MOVE_STATUS_SIZE : Word := 16#8483;   // MOVE_BLK_VARIANT: DEST too small
      FB_STATE_NO_PROCESSING : USInt := 0;   // FB state: No processing
      FB_STATE_INIT : USInt := 1;   // FB state: initialization
      FB_STATE_REQUEST : USInt := 2;   // FB state: prepare request
      FB_STATE_SEND : USInt := 3;   // FB state: send request
      FB_STATE_RCV : USInt := 4;   // FB state: receive data
      FB_STATE_MON : USInt := 5;   // FB state: monitoring connection
      CRLF : String := '$R$L';   // Newline control character (carriage return, line feed)
      HEADER_END : String := '$R$L$R$L';   // End of HTTP header (two newline control characters)
      LEN_CRLF : UInt := 2;   // Length of CRLF
      SCHEME_HTTP : String := 'http://';   // Scheme HTTP
      SCHEME_HTTPS : String := 'https://';   // Scheme HTTPS
   END_VAR
   // statParam.paramIP.ConnPara.ActiveEstablished := true;
   // statParam.paramQDN.ConnPara.ActiveEstablished := true;
BEGIN
   REGION BLOCK INFO HEADER
     //===============================================================================
     // SIEMENS / (c)Copyright 2024
     //-------------------------------------------------------------------------------
     // Title:        LHTTP_Get
     // Function:     Implements the HTTP GET method
     // Library:      LHTTP
     // Author:       Siemens Industry Online Support
     // Tested with:  CPU 1516-3 PN/DP V2.9
     // Engineering:  TIA Portal V17
     // Restrictions: --
     // Requirements: S7-1200 with firmware V4.4 or higher
     //               S7-1500 with firmware V2.0 or higher
     //-------------------------------------------------------------------------------
     // Change log table:
     // Version  | Date       | Expert in charge       | Changes applied
     //----------|------------|------------------------|------------------------------
     // 02.02.00 | 2024-04-05 | Online Support         | Changed behavior that HTTPS is used by default
     //          |            |                        | Improved evaluation of host in URL
     //----------|------------|------------------------|------------------------------
     // 02.01.04 | 2023-08-23 | Online Support         | Fixed issue when first packet of response only contains header or response header is not received completely in one packet
     //----------|------------|------------------------|------------------------------
     // 02.01.01 | 2023-02-23 | Online Support         | Changed data type of "statContentLength" to allow larger content size
     //----------|------------|------------------------|------------------------------
     // 02.01.00 | 2021-12-15 | Online Support         | Renamed parameter "data" to "queryParams"
     //-------------------------------------------------------------------------------
     // 02.00.04 | 2021-05-10 | Online Support         | Fixed issues with chunked encoding
     //          |            |                        | Allow chunk sizes > 65535 Bytes
     //          |            |                        | Made header evaluation case-insensitive
     //-------------------------------------------------------------------------------
     // 02.00.00 | 2020-12-16 | Online Support         | Added option to keep connection established
     //          |            |                        | Added parameter to add user-defined headers fields
     //          |            |                        | Changed to data type of "data" to Variant to allow larger data
     //          |            |                        | Removed "statusID" and added "diagnostics" instead, changed some error codes
     //-------------------------------------------------------------------------------
     // 01.00.00 | 2019-04-01 | Online Support         | First released version
     //===============================================================================
   END_REGION

   REGION INSTRUCTIONS
     IF (#statStatus <> #STATUS_IDLE) THEN // Only execute when FB is triggered to reduce system load
       // Connect and send
       IF #statParam.isQDN THEN // Call if host is a domain name
         #instTSendC(REQ     := #statSend.req,
                     CONT    := #statSend.connect,
                     LEN     := #statRequest.length,
                     CONNECT := #statParam.paramQDN,
                     DATA    := #statRequest.chars);
       ELSE // Call if host is an IP address
         #instTSendC(REQ     := #statSend.req,
                     CONT    := #statSend.connect,
                     LEN     := #statRequest.length,
                     CONNECT := #statParam.paramIP,
                     DATA    := #statRequest.chars);
       END_IF;

       // Receive
       #instTRcv(ID    := #statParam.paramQDN.ConnPara.ID,
                 EN_R  := #statFBState >= #FB_STATE_RCV,
                 LEN   := 0,
                 ADHOC := true,
                 DATA  := #statRcvBuffer);

       // Monitor time out
       #instTimeout(IN := #statTimeoutIn,
                    PT := #timeOut);

       IF #instTimeout.Q THEN
         #statStatus := #ERR_TIMEOUT;
       END_IF;
     END_IF;
   END_REGION

   REGION TRIGGERING
     IF (#execute = true AND #statExecuteOld = false) // Check if FB is triggered
       AND (#statStatus = #STATUS_IDLE OR #statStatus = #STATUS_MONITORING)
     THEN // First call; initialize FB
       // Copy URL
       #tempUrl := #url;

       #statBusy := true;
       #statStatus := #STATUS_FIRST_CALL;
       #statSubfunctionStatus := #SUB_STATUS_NO_ERROR;
       #diagnostics := #statEmptyDiagnostics;

       IF #statConnected = FALSE THEN // Connection is not yet established
         #statFBState := #FB_STATE_INIT;
       ELSE // Connection is already established, skip init
         #statFBState := #FB_STATE_REQUEST;
       END_IF;

     ELSIF (#statStatus = #STATUS_FIRST_CALL) THEN
       #statStatus := #STATUS_CONNECTING;
     END_IF;

     // Edge detection 'execute' input
     #statExecuteOld := #execute;
   END_REGION TRIGGERING

   IF (#statStatus = #STATUS_IDLE) THEN // Nothing to do -> End here to reduce "system load"
     RETURN;
   END_IF;

   REGION STATE_MACHINE
     // State machine is wrapped in REPEAT loop to make it possible to quickly exit state machine
     // in case of an error or to go through CASE multiple times within one cycle
     REPEAT
       #tempExitLoop := true; // Condition to exit loop is set per default

       CASE #statFBState OF // State machine of FB
         #FB_STATE_NO_PROCESSING: // No processing active
           ;

         #FB_STATE_INIT:
           REGION INIT
             // Get size of receive buffer
             IF LOWER_BOUND(ARR := #responseData, DIM := 1) <> 0 THEN
               #statStatus := #ERR_BOUND_NOT_ZERO;
               EXIT;
             ELSE
               #statSizeRcvArray := DINT_TO_UDINT(UPPER_BOUND(ARR := #responseData, DIM := 1)) + 1;
             END_IF;

             // Set connection parameters
             #statParam.paramQDN.ConnPara.InterfaceId := #hwID;
             #statParam.paramQDN.ConnPara.ID := #connID;
             #statParam.paramIP.ConnPara.InterfaceId := #hwID;
             #statParam.paramIP.ConnPara.ID := #connID;

             // Check if 'http' was explicitely specified for connection to be unsecure
             IF LEFT(IN := #tempUrl, L := LEN(#SCHEME_HTTP)) = #SCHEME_HTTP THEN // HTTP
               #statParam.paramQDN.ActivateSecureConn := false;
               #statParam.paramIP.ActivateSecureConn := false;
               #tempUrl := DELETE(IN := #tempUrl, L := LEN(#SCHEME_HTTP), P := 1); // Delete network protocol from URL
             ELSE // HTTPS
               #statParam.paramQDN.ActivateSecureConn := true;
               #statParam.paramQDN.ExtTLSCapabilities.%X0 := #tls.validateServerIdentity;
               #statParam.paramQDN.TLSServerCertRef := #tls.serverCert;
               #statParam.paramQDN.TLSClientCertRef := #tls.clientCert;
               #statParam.paramIP.ActivateSecureConn := true;
               #statParam.paramIP.ExtTLSCapabilities.%X0 := #tls.validateServerIdentity;
               #statParam.paramIP.TLSServerCertRef := #tls.serverCert;
               #statParam.paramIP.TLSClientCertRef := #tls.clientCert;

               // Delete network protocol from URL if specified
               IF LEFT(IN := #tempUrl, L := LEN(#SCHEME_HTTPS)) = #SCHEME_HTTPS THEN
                 #tempUrl := DELETE(IN := #tempUrl, L := LEN(#SCHEME_HTTPS), P := 1);
               END_IF;
             END_IF;

             // Get host name and port
             #tempPos := FIND(IN1 := #tempUrl, IN2 := '/');
             IF #tempPos > 0 THEN // URL has a path after host name
               #statHost := LEFT(IN := #tempUrl, L := #tempPos - 1); // Strip path
             ELSE
               #statHost := #tempUrl;
             END_IF;

             #tempPos := FIND(IN1 := #statHost, IN2 := ':');
             IF #tempPos > 0 THEN // Port specified in URL
               #statParam.paramQDN.ConnPara.RemotePort := STRING_TO_UINT(DELETE(IN := #statHost, L := #tempPos, P := 1));
               #statParam.paramIP.ConnPara.RemotePort := STRING_TO_UINT(DELETE(IN := #statHost, L := #tempPos, P := 1));
               #statHost := LEFT(IN := #statHost, L := #tempPos - 1); // Strip port
             ELSE // No port specified in URL, set default port
               IF #statParam.paramQDN.ActivateSecureConn OR #statParam.paramIP.ActivateSecureConn THEN
                 #statParam.paramQDN.ConnPara.RemotePort := #PORT_SECURE;
                 #statParam.paramIP.ConnPara.RemotePort := #PORT_SECURE;
               ELSE
                 #statParam.paramQDN.ConnPara.RemotePort := #PORT_UNSECURE;
                 #statParam.paramIP.ConnPara.RemotePort := #PORT_UNSECURE;
               END_IF;
             END_IF;

